LIN {X 0,Y 312.483,Z 284.187,A -85,B 0,C 180,E1 -15707.917,E2 -15707.917} C_VEL
LIN {X 0,Y 312.533,Z 284.181,A -85,B 0,C 180,E1 -15711.909,E2 -15711.909} C_VEL
LIN {X 0,Y 312.504,Z 284.186,A -85,B 0,C 180,E1 -15715.788,E2 -15715.788} C_VEL
LIN {X 0,Y 312.503,Z 284.18,A -85,B 0,C 180,E1 -15718.85,E2 -15718.85} C_VEL
LIN {X 0,Y 312.537,Z 284.181,A -85,B 0,C 180,E1 -15721.82,E2 -15721.82} C_VEL
LIN {X 0,Y 312.544,Z 284.175,A -85,B 0,C 180,E1 -15724.706,E2 -15724.706} C_VEL
LIN {X 0,Y 312.559,Z 284.177,A -85,B 0,C 180,E1 -15727.525,E2 -15727.525} C_VEL
LIN {X 0,Y 312.562,Z 284.179,A -85,B 0,C 180,E1 -15731.65,E2 -15731.65} C_VEL
LIN {X 0,Y 312.68,Z 284.164,A -85,B 0,C 180,E1 -15735.684,E2 -15735.684} C_VEL
LIN {X 0,Y 312.696,Z 284.162,A -85,B 0,C 180,E1 -15739.64,E2 -15739.64} C_VEL
LIN {X 0,Y 312.865,Z 284.136,A -85,B 0,C 180,E1 -15742.252,E2 -15742.252} C_VEL
LIN {X 0,Y 312.708,Z 284.155,A -85,B 0,C 180,E1 -15744.841,E2 -15744.841} C_VEL
LIN {X 0,Y 312.982,Z 284.121,A -85,B 0,C 180,E1 -15748.712,E2 -15748.712} C_VEL
LIN {X 0,Y 312.982,Z 284.123,A -85,B 0,C 180,E1 -15751.285,E2 -15751.285} C_VEL
LIN {X 0,Y 312.707,Z 284.157,A -85,B 0,C 180,E1 -15755.156,E2 -15755.156} C_VEL
LIN {X 0,Y 312.862,Z 284.139,A -85,B 0,C 180,E1 -15757.744,E2 -15757.744} C_VEL
LIN {X 0,Y 312.659,Z 284.164,A -85,B 0,C 180,E1 -15761.67,E2 -15761.67} C_VEL
LIN {X 0,Y 312.69,Z 284.158,A -85,B 0,C 180,E1 -15764.886,E2 -15764.886} C_VEL
LIN {X 0,Y 312.619,Z 284.169,A -85,B 0,C 180,E1 -15769.235,E2 -15769.235} C_VEL
LIN {X 0,Y 312.535,Z 284.177,A -85,B 0,C 180,E1 -15772.788,E2 -15772.788} C_VEL
LIN {X 0,Y 312.585,Z 284.171,A -85,B 0,C 180,E1 -15775.932,E2 -15775.932} C_VEL
LIN {X 0,Y 312.526,Z 284.18,A -85,B 0,C 180,E1 -15779.65,E2 -15779.65} C_VEL
LIN {X 0,Y 312.507,Z 284.182,A -85,B 0,C 180,E1 -15783.688,E2 -15783.688} C_VEL
LIN {X 0,Y 312.525,Z 284.183,A -85,B 0,C 180,E1 -15787.383,E2 -15787.383} C_VEL
LIN {X 0,Y 312.477,Z 284.184,A -85,B 0,C 180,E1 -15790.708,E2 -15790.708} C_VEL
LIN {X 0,Y 312.459,Z 284.185,A -85,B 0,C 180,E1 -15794.205,E2 -15794.205} C_VEL
LIN {X 0,Y 312.472,Z 284.185,A -85,B 0,C 180,E1 -15797.918,E2 -15797.918} C_VEL
LIN {X 0,Y 312.491,Z 284.182,A -85,B 0,C 180,E1 -15801.917,E2 -15801.917} C_VEL
LIN {X 0,Y 312.517,Z 284.178,A -85,B 0,C 180,E1 -15804.22,E2 -15804.22} C_VEL
LIN {X 0,Y 312.49,Z 284.186,A -85,B 0,C 180,E1 -15807.334,E2 -15807.334} C_VEL
LIN {X 0,Y 312.538,Z 284.18,A -85,B 0,C 180,E1 -15811.276,E2 -15811.276} C_VEL
LIN {X 0,Y 312.541,Z 284.176,A -85,B 0,C 180,E1 -15812.722,E2 -15812.722} C_VEL
LIN {X 0,Y 311.9,Z 284.261,A -85,B 0,C 180,E1 -15813.797,E2 -15813.797} C_VEL
LIN {X 0,Y 309.062,Z 284.619,A -85,B 0,C 180,E1 -15815.546,E2 -15815.546} C_VEL
LIN {X 0,Y 306.628,Z 284.92,A -85,B 0,C 180,E1 -15816.965,E2 -15816.965} C_VEL
LIN {X 0,Y 305.562,Z 285.047,A -85,B 0,C 180,E1 -15818.063,E2 -15818.063} C_VEL
LIN {X 0,Y 305.466,Z 285.057,A -85,B 0,C 180,E1 -15818.435,E2 -15818.435} C_VEL
LIN {X 0,Y 305.566,Z 285.049,A -85,B 0,C 180,E1 -15821.217,E2 -15821.217} C_VEL
LIN {X 0,Y 305.635,Z 285.039,A -85,B 0,C 180,E1 -15825.35,E2 -15825.35} C_VEL
LIN {X 0,Y 305.625,Z 285.04,A -85,B 0,C 180,E1 -15829.4,E2 -15829.4} C_VEL
LIN {X 0,Y 305.795,Z 285.016,A -85,B 0,C 180,E1 -15832.075,E2 -15832.075} C_VEL
LIN {X 0,Y 305.673,Z 285.033,A -85,B 0,C 180,E1 -15834.724,E2 -15834.724} C_VEL
LIN {X 0,Y 305.945,Z 284.999,A -85,B 0,C 180,E1 -15838.685,E2 -15838.685} C_VEL
LIN {X 0,Y 305.946,Z 285,A -85,B 0,C 180,E1 -15841.317,E2 -15841.317} C_VEL
LIN {X 0,Y 305.84,Z 285.012,A -85,B 0,C 180,E1 -15846.599,E2 -15846.599} C_VEL
LIN {X 0,Y 305.725,Z 285.027,A -85,B 0,C 180,E1 -15849.261,E2 -15849.261} C_VEL
LIN {X 0,Y 305.578,Z 285.045,A -85,B 0,C 180,E1 -15853.297,E2 -15853.297} C_VEL
LIN {X 0,Y 305.583,Z 285.042,A -85,B 0,C 180,E1 -15856.022,E2 -15856.022} C_VEL
LIN {X 0,Y 305.55,Z 285.048,A -85,B 0,C 180,E1 -15859.438,E2 -15859.438} C_VEL
LIN {X 0,Y 305.476,Z 285.06,A -85,B 0,C 180,E1 -15863.041,E2 -15863.041} C_VEL
LIN {X 0,Y 305.517,Z 285.052,A -85,B 0,C 180,E1 -15866.221,E2 -15866.221} C_VEL
LIN {X 0,Y 305.487,Z 285.058,A -85,B 0,C 180,E1 -15869.052,E2 -15869.052} C_VEL
LIN {X 0,Y 305.457,Z 285.059,A -85,B 0,C 180,E1 -15873.519,E2 -15873.519} C_VEL
LIN {X 0,Y 305.464,Z 285.062,A -85,B 0,C 180,E1 -15876.742,E2 -15876.742} C_VEL
LIN {X 0,Y 305.448,Z 285.063,A -85,B 0,C 180,E1 -15880.602,E2 -15880.602} C_VEL
LIN {X 0,Y 305.413,Z 285.066,A -85,B 0,C 180,E1 -15884.495,E2 -15884.495} C_VEL
LIN {X 0,Y 305.439,Z 285.062,A -85,B 0,C 180,E1 -15888.146,E2 -15888.146} C_VEL
LIN {X 0,Y 305.483,Z 285.18,A -85,B 0,C 180,E1 -15889.323,E2 -15889.323} C_VEL
LIN {X 0,Y 309.162,Z 300.003,A -85,B 0,C 180,E1 -15893.056,E2 -15893.056} C_VEL
LIN {X 0,Y 311.75,Z 310.492,A -85,B 0,C 180,E1 -15895.574,E2 -15895.574} C_VEL
LIN {X 0,Y 318.467,Z 328.782,A -85,B 0,C 180,E1 -15896.765,E2 -15896.765} C_VEL
LIN {X 0,Y 323.204,Z 363.617,A -85,B 0,C 180,E1 -15898.341,E2 -15898.341} C_VEL
LIN {X 0,Y 317.418,Z 478.074,A -85,B 0,C 180,E1 -15901.98,E2 -15901.98} C_VEL
LIN {X 0,Y 316.163,Z 494.683,A -85,B 0,C 180,E1 -15902.769,E2 -15902.769} C_VEL
LIN {X 0,Y 314.676,Z 509.82,A -85,B 0,C 180,E1 -15903.739,E2 -15903.739} C_VEL
LIN {X 0,Y 313.128,Z 524.404,A -85,B 0,C 180,E1 -15904.938,E2 -15904.938} C_VEL
LIN {X 0,Y 311.443,Z 538.622,A -85,B 0,C 180,E1 -15906.39,E2 -15906.39} C_VEL
LIN {X 0,Y 309.762,Z 551.702,A -85,B 0,C 180,E1 -15908.018,E2 -15908.018} C_VEL
LIN {X 0,Y 308.306,Z 563.036,A -85,B 0,C 180,E1 -15909.703,E2 -15909.703} C_VEL
LIN {X 0,Y 306.969,Z 574.069,A -85,B 0,C 180,E1 -15911.653,E2 -15911.653} C_VEL
LIN {X 0,Y 305.696,Z 585.036,A -85,B 0,C 180,E1 -15913.987,E2 -15913.987} C_VEL
LIN {X 0,Y 304.836,Z 594.132,A -85,B 0,C 180,E1 -15916.341,E2 -15916.341} C_VEL
LIN {X 0,Y 304.283,Z 601.551,A -85,B 0,C 180,E1 -15918.68,E2 -15918.68} C_VEL
LIN {X 0,Y 303.985,Z 608.343,A -85,B 0,C 180,E1 -15921.359,E2 -15921.359} C_VEL
LIN {X 0,Y 303.954,Z 613.202,A -85,B 0,C 180,E1 -15923.854,E2 -15923.854} C_VEL
LIN {X 0,Y 303.841,Z 616.375,A -85,B 0,C 180,E1 -15926.023,E2 -15926.023} C_VEL
LIN {X 0,Y 304.058,Z 618.937,A -85,B 0,C 180,E1 -15928.677,E2 -15928.677} C_VEL
LIN {X 0,Y 304.045,Z 619.678,A -85,B 0,C 180,E1 -15930.002,E2 -15930.002} C_VEL
LIN {X 0,Y 303.957,Z 620.077,A -85,B 0,C 180,E1 -15931.327,E2 -15931.327} C_VEL
LIN {X 0,Y 303.763,Z 619.886,A -85,B 0,C 180,E1 -15933.982,E2 -15933.982} C_VEL
LIN {X 0,Y 303.706,Z 618.409,A -85,B 0,C 180,E1 -15936.646,E2 -15936.646} C_VEL
LIN {X 0,Y 303.899,Z 615.68,A -85,B 0,C 180,E1 -15939.318,E2 -15939.318} C_VEL
LIN {X 0,Y 304.501,Z 611.675,A -85,B 0,C 180,E1 -15941.991,E2 -15941.991} C_VEL
LIN {X 0,Y 305.543,Z 606.341,A -85,B 0,C 180,E1 -15944.658,E2 -15944.658} C_VEL
LIN {X 0,Y 307.205,Z 599.572,A -85,B 0,C 180,E1 -15947.303,E2 -15947.303} C_VEL
LIN {X 0,Y 309.461,Z 591.258,A -85,B 0,C 180,E1 -15949.919,E2 -15949.919} C_VEL
LIN {X 0,Y 311.889,Z 582.568,A -85,B 0,C 180,E1 -15952.177,E2 -15952.177} C_VEL
LIN {X 0,Y 315.026,Z 572.349,A -85,B 0,C 180,E1 -15954.378,E2 -15954.378} C_VEL
LIN {X 0,Y 318.596,Z 560.378,A -85,B 0,C 180,E1 -15956.534,E2 -15956.534} C_VEL
LIN {X 0,Y 322.495,Z 547.288,A -85,B 0,C 180,E1 -15958.473,E2 -15958.473} C_VEL
LIN {X 0,Y 326.441,Z 533.561,A -85,B 0,C 180,E1 -15960.143,E2 -15960.143} C_VEL
LIN {X 0,Y 330.508,Z 518.79,A -85,B 0,C 180,E1 -15961.599,E2 -15961.599} C_VEL
LIN {X 0,Y 334.241,Z 504,A -85,B 0,C 180,E1 -15962.783,E2 -15962.783} C_VEL
LIN {X 0,Y 337.95,Z 487.774,A -85,B 0,C 180,E1 -15963.801,E2 -15963.801} C_VEL
LIN {X 0,Y 341.362,Z 470.013,A -85,B 0,C 180,E1 -15964.664,E2 -15964.664} C_VEL
LIN {X 0,Y 353.831,Z 389.949,A -85,B 0,C 180,E1 -15967.737,E2 -15967.737} C_VEL
LIN {X 0,Y 357.008,Z 371.451,A -85,B 0,C 180,E1 -15968.451,E2 -15968.451} C_VEL
LIN {X 0,Y 357.448,Z 364.254,A -85,B 0,C 180,E1 -15969.081,E2 -15969.081} C_VEL
LIN {X 0,Y 356.3,Z 359.523,A -85,B 0,C 180,E1 -15970.263,E2 -15970.263} C_VEL
LIN {X 0,Y 355.233,Z 355.391,A -85,B 0,C 180,E1 -15971.627,E2 -15971.627} C_VEL
LIN {X 0,Y 354.276,Z 351.159,A -85,B 0,C 180,E1 -15973.708,E2 -15973.708} C_VEL
LIN {X 0,Y 354.116,Z 349.484,A -85,B 0,C 180,E1 -15975.187,E2 -15975.187} C_VEL
LIN {X 0,Y 354.487,Z 349.334,A -85,B 0,C 180,E1 -15977.187,E2 -15977.187} C_VEL
LIN {X 0,Y 355.969,Z 350.738,A -85,B 0,C 180,E1 -15979.342,E2 -15979.342} C_VEL
LIN {X 0,Y 357.608,Z 353.477,A -85,B 0,C 180,E1 -15980.911,E2 -15980.911} C_VEL
LIN {X 0,Y 358.995,Z 356.175,A -85,B 0,C 180,E1 -15981.975,E2 -15981.975} C_VEL
LIN {X 0,Y 347.517,Z 422.744,A -85,B 0,C 180,E1 -15984.537,E2 -15984.537} C_VEL
LIN {X 0,Y 342.784,Z 453.541,A -85,B 0,C 180,E1 -15985.767,E2 -15985.767} C_VEL
LIN {X 0,Y 339.824,Z 469.984,A -85,B 0,C 180,E1 -15986.677,E2 -15986.677} C_VEL
LIN {X 0,Y 336.515,Z 485.723,A -85,B 0,C 180,E1 -15987.821,E2 -15987.821} C_VEL
LIN {X 0,Y 333.231,Z 499.427,A -85,B 0,C 180,E1 -15989.063,E2 -15989.063} C_VEL
LIN {X 0,Y 329.525,Z 513.47,A -85,B 0,C 180,E1 -15990.623,E2 -15990.623} C_VEL
LIN {X 0,Y 325.894,Z 525.991,A -85,B 0,C 180,E1 -15992.318,E2 -15992.318} C_VEL
LIN {X 0,Y 322.284,Z 537.29,A -85,B 0,C 180,E1 -15994.142,E2 -15994.142} C_VEL
LIN {X 0,Y 318.668,Z 548.098,A -85,B 0,C 180,E1 -15996.265,E2 -15996.265} C_VEL
LIN {X 0,Y 315.639,Z 557.162,A -85,B 0,C 180,E1 -15998.445,E2 -15998.445} C_VEL
LIN {X 0,Y 312.714,Z 565.295,A -85,B 0,C 180,E1 -16000.805,E2 -16000.805} C_VEL
LIN {X 0,Y 310.44,Z 571.206,A -85,B 0,C 180,E1 -16002.883,E2 -16002.883} C_VEL
LIN {X 0,Y 308.415,Z 577.037,A -85,B 0,C 180,E1 -16005.482,E2 -16005.482} C_VEL
LIN {X 0,Y 306.824,Z 581.492,A -85,B 0,C 180,E1 -16008.102,E2 -16008.102} C_VEL
LIN {X 0,Y 305.638,Z 584.662,A -85,B 0,C 180,E1 -16010.736,E2 -16010.736} C_VEL
LIN {X 0,Y 304.678,Z 586.616,A -85,B 0,C 180,E1 -16013.376,E2 -16013.376} C_VEL
LIN {X 0,Y 304.271,Z 587.337,A -85,B 0,C 180,E1 -16016.026,E2 -16016.026} C_VEL
LIN {X 0,Y 303.995,Z 586.847,A -85,B 0,C 180,E1 -16018.674,E2 -16018.674} C_VEL
LIN {X 0,Y 303.845,Z 585.118,A -85,B 0,C 180,E1 -16021.324,E2 -16021.324} C_VEL
LIN {X 0,Y 303.946,Z 582.089,A -85,B 0,C 180,E1 -16023.977,E2 -16023.977} C_VEL
LIN {X 0,Y 304.108,Z 577.7,A -85,B 0,C 180,E1 -16026.634,E2 -16026.634} C_VEL
LIN {X 0,Y 304.48,Z 571.858,A -85,B 0,C 180,E1 -16029.297,E2 -16029.297} C_VEL
LIN {X 0,Y 305.091,Z 564.369,A -85,B 0,C 180,E1 -16031.964,E2 -16031.964} C_VEL
LIN {X 0,Y 306.037,Z 556.302,A -85,B 0,C 180,E1 -16034.291,E2 -16034.291} C_VEL
LIN {X 0,Y 307.118,Z 546.548,A -85,B 0,C 180,E1 -16036.62,E2 -16036.62} C_VEL
LIN {X 0,Y 308.375,Z 536.618,A -85,B 0,C 180,E1 -16038.605,E2 -16038.605} C_VEL
LIN {X 0,Y 309.868,Z 524.859,A -85,B 0,C 180,E1 -16040.581,E2 -16040.581} C_VEL
LIN {X 0,Y 311.38,Z 512.154,A -85,B 0,C 180,E1 -16042.363,E2 -16042.363} C_VEL
LIN {X 0,Y 312.995,Z 497.882,A -85,B 0,C 180,E1 -16044.014,E2 -16044.014} C_VEL
LIN {X 0,Y 314.43,Z 484.235,A -85,B 0,C 180,E1 -16045.306,E2 -16045.306} C_VEL
LIN {X 0,Y 315.759,Z 469.495,A -85,B 0,C 180,E1 -16046.431,E2 -16046.431} C_VEL
LIN {X 0,Y 316.948,Z 453.178,A -85,B 0,C 180,E1 -16047.392,E2 -16047.392} C_VEL
LIN {X 0,Y 317.883,Z 437.277,A -85,B 0,C 180,E1 -16048.065,E2 -16048.065} C_VEL
LIN {X 0,Y 323.396,Z 326.411,A -85,B 0,C 180,E1 -16051.547,E2 -16051.547} C_VEL
LIN {X 0,Y 307.407,Z 290.038,A -85,B 0,C 180,E1 -16054.103,E2 -16054.103} C_VEL
LIN {X 0,Y 305.517,Z 285.343,A -85,B 0,C 180,E1 -16054.439,E2 -16054.439} C_VEL
LIN {X 0,Y 305.491,Z 285.056,A -85,B 0,C 180,E1 -16054.482,E2 -16054.482} C_VEL
LIN {X 0,Y 305.427,Z 285.063,A -85,B 0,C 180,E1 -16058.521,E2 -16058.521} C_VEL
LIN {X 0,Y 305.439,Z 285.066,A -85,B 0,C 180,E1 -16061.855,E2 -16061.855} C_VEL
LIN {X 0,Y 305.399,Z 285.068,A -85,B 0,C 180,E1 -16065.509,E2 -16065.509} C_VEL
LIN {X 0,Y 305.44,Z 285.063,A -85,B 0,C 180,E1 -16068.141,E2 -16068.141} C_VEL
LIN {X 0,Y 305.493,Z 285.057,A -85,B 0,C 180,E1 -16071.598,E2 -16071.598} C_VEL
LIN {X 0,Y 305.46,Z 285.058,A -85,B 0,C 180,E1 -16074.885,E2 -16074.885} C_VEL
LIN {X 0,Y 305.438,Z 285.061,A -85,B 0,C 180,E1 -16078.356,E2 -16078.356} C_VEL
LIN {X 0,Y 305.482,Z 285.056,A -85,B 0,C 180,E1 -16081.108,E2 -16081.108} C_VEL
LIN {X 0,Y 305.497,Z 285.055,A -85,B 0,C 180,E1 -16084.08,E2 -16084.08} C_VEL
LIN {X 0,Y 305.488,Z 285.055,A -85,B 0,C 180,E1 -16086.975,E2 -16086.975} C_VEL
LIN {X 0,Y 305.513,Z 285.053,A -85,B 0,C 180,E1 -16091.211,E2 -16091.211} C_VEL
LIN {X 0,Y 305.621,Z 285.041,A -85,B 0,C 180,E1 -16095.346,E2 -16095.346} C_VEL
LIN {X 0,Y 305.632,Z 285.04,A -85,B 0,C 180,E1 -16099.398,E2 -16099.398} C_VEL
LIN {X 0,Y 305.806,Z 285.016,A -85,B 0,C 180,E1 -16102.072,E2 -16102.072} C_VEL
LIN {X 0,Y 305.68,Z 285.03,A -85,B 0,C 180,E1 -16104.722,E2 -16104.722} C_VEL
LIN {X 0,Y 305.949,Z 284.997,A -85,B 0,C 180,E1 -16108.682,E2 -16108.682} C_VEL
LIN {X 0,Y 305.949,Z 285,A -85,B 0,C 180,E1 -16111.314,E2 -16111.314} C_VEL
LIN {X 0,Y 305.843,Z 285.01,A -85,B 0,C 180,E1 -16116.596,E2 -16116.596} C_VEL
LIN {X 0,Y 305.727,Z 285.027,A -85,B 0,C 180,E1 -16119.258,E2 -16119.258} C_VEL
LIN {X 0,Y 305.579,Z 285.046,A -85,B 0,C 180,E1 -16123.294,E2 -16123.294} C_VEL
LIN {X 0,Y 305.583,Z 285.043,A -85,B 0,C 180,E1 -16126.019,E2 -16126.019} C_VEL
LIN {X 0,Y 305.566,Z 285.049,A -85,B 0,C 180,E1 -16129.443,E2 -16129.443} C_VEL
LIN {X 0,Y 305.479,Z 285.057,A -85,B 0,C 180,E1 -16133.04,E2 -16133.04} C_VEL
LIN {X 0,Y 305.514,Z 285.051,A -85,B 0,C 180,E1 -16136.217,E2 -16136.217} C_VEL
LIN {X 0,Y 305.476,Z 285.058,A -85,B 0,C 180,E1 -16139.046,E2 -16139.046} C_VEL
LIN {X 0,Y 305.429,Z 285.062,A -85,B 0,C 180,E1 -16141.951,E2 -16141.951} C_VEL
LIN {X 0,Y 305.45,Z 285.062,A -85,B 0,C 180,E1 -16145.112,E2 -16145.112} C_VEL
LIN {X 0,Y 305.436,Z 285.061,A -85,B 0,C 180,E1 -16148.528,E2 -16148.528} C_VEL
LIN {X 0,Y 305.446,Z 285.06,A -85,B 0,C 180,E1 -16152.586,E2 -16152.586} C_VEL
LIN {X 0,Y 305.429,Z 285.061,A -85,B 0,C 180,E1 -16156.347,E2 -16156.347} C_VEL
LIN {X 0,Y 305.444,Z 285.06,A -85,B 0,C 180,E1 -16159.892,E2 -16159.892} C_VEL
LIN {X 0,Y 305.467,Z 285.059,A -85,B 0,C 180,E1 -16163.631,E2 -16163.631} C_VEL
LIN {X 0,Y 305.451,Z 285.059,A -85,B 0,C 180,E1 -16166.483,E2 -16166.483} C_VEL
LIN {X 0,Y 305.482,Z 285.058,A -85,B 0,C 180,E1 -16170.95,E2 -16170.95} C_VEL
LIN {X 0,Y 305.558,Z 285.045,A -85,B 0,C 180,E1 -16174.088,E2 -16174.088} C_VEL
LIN {X 0,Y 305.466,Z 285.057,A -85,B 0,C 180,E1 -16178.435,E2 -16178.435} C_VEL
LIN {X 0,Y 304.775,Z 285.145,A -85,B 0,C 180,E1 -16179.537,E2 -16179.537} C_VEL
LIN {X 0,Y 301.943,Z 285.499,A -85,B 0,C 180,E1 -16181.332,E2 -16181.332} C_VEL
LIN {X 0,Y 299.585,Z 285.792,A -85,B 0,C 180,E1 -16182.788,E2 -16182.788} C_VEL
LIN {X 0,Y 298.613,Z 285.911,A -85,B 0,C 180,E1 -16183.915,E2 -16183.915} C_VEL
LIN {X 0,Y 298.553,Z 285.918,A -85,B 0,C 180,E1 -16184.296,E2 -16184.296} C_VEL
LIN {X 0,Y 298.54,Z 285.919,A -85,B 0,C 180,E1 -16187.769,E2 -16187.769} C_VEL
LIN {X 0,Y 298.741,Z 285.895,A -85,B 0,C 180,E1 -16191.887,E2 -16191.887} C_VEL
LIN {X 0,Y 298.644,Z 285.908,A -85,B 0,C 180,E1 -16194.6,E2 -16194.6} C_VEL
LIN {X 0,Y 298.911,Z 285.875,A -85,B 0,C 180,E1 -16198.654,E2 -16198.654} C_VEL
LIN {X 0,Y 298.913,Z 285.875,A -85,B 0,C 180,E1 -16201.348,E2 -16201.348} C_VEL
LIN {X 0,Y 298.785,Z 285.892,A -85,B 0,C 180,E1 -16206.755,E2 -16206.755} C_VEL
LIN {X 0,Y 298.67,Z 285.905,A -85,B 0,C 180,E1 -16209.482,E2 -16209.482} C_VEL
LIN {X 0,Y 298.541,Z 285.92,A -85,B 0,C 180,E1 -16213.617,E2 -16213.617} C_VEL
LIN {X 0,Y 298.538,Z 285.921,A -85,B 0,C 180,E1 -16216.41,E2 -16216.41} C_VEL
LIN {X 0,Y 298.488,Z 285.927,A -85,B 0,C 180,E1 -16219.649,E2 -16219.649} C_VEL
LIN {X 0,Y 298.419,Z 285.936,A -85,B 0,C 180,E1 -16223.602,E2 -16223.602} C_VEL
LIN {X 0,Y 298.477,Z 285.931,A -85,B 0,C 180,E1 -16226.577,E2 -16226.577} C_VEL
LIN {X 0,Y 298.412,Z 285.936,A -85,B 0,C 180,E1 -16229.643,E2 -16229.643} C_VEL
LIN {X 0,Y 298.387,Z 285.944,A -85,B 0,C 180,E1 -16232.802,E2 -16232.802} C_VEL
LIN {X 0,Y 298.436,Z 285.938,A -85,B 0,C 180,E1 -16236.809,E2 -16236.809} C_VEL
LIN {X 0,Y 298.381,Z 285.942,A -85,B 0,C 180,E1 -16241.09,E2 -16241.09} C_VEL
LIN {X 0,Y 298.383,Z 285.942,A -85,B 0,C 180,E1 -16245.044,E2 -16245.044} C_VEL
LIN {X 0,Y 298.417,Z 286.041,A -85,B 0,C 180,E1 -16248.854,E2 -16248.854} C_VEL
LIN {X 0,Y 302.253,Z 301.368,A -85,B 0,C 180,E1 -16252.806,E2 -16252.806} C_VEL
LIN {X 0,Y 304.389,Z 310.097,A -85,B 0,C 180,E1 -16254.948,E2 -16254.948} C_VEL
LIN {X 0,Y 312.03,Z 331.055,A -85,B 0,C 180,E1 -16256.362,E2 -16256.362} C_VEL
LIN {X 0,Y 316.55,Z 364.738,A -85,B 0,C 180,E1 -16257.919,E2 -16257.919} C_VEL
LIN {X 0,Y 310.599,Z 477.927,A -85,B 0,C 180,E1 -16261.632,E2 -16261.632} C_VEL
LIN {X 0,Y 309.42,Z 493.04,A -85,B 0,C 180,E1 -16262.354,E2 -16262.354} C_VEL
LIN {X 0,Y 307.855,Z 508.932,A -85,B 0,C 180,E1 -16263.386,E2 -16263.386} C_VEL
LIN {X 0,Y 306.165,Z 524.431,A -85,B 0,C 180,E1 -16264.691,E2 -16264.691} C_VEL
LIN {X 0,Y 304.46,Z 538.557,A -85,B 0,C 180,E1 -16266.176,E2 -16266.176} C_VEL
LIN {X 0,Y 302.736,Z 551.563,A -85,B 0,C 180,E1 -16267.839,E2 -16267.839} C_VEL
LIN {X 0,Y 301.165,Z 563.609,A -85,B 0,C 180,E1 -16269.691,E2 -16269.691} C_VEL
LIN {X 0,Y 299.892,Z 573.843,A -85,B 0,C 180,E1 -16271.558,E2 -16271.558} C_VEL
LIN {X 0,Y 298.631,Z 584.784,A -85,B 0,C 180,E1 -16273.949,E2 -16273.949} C_VEL
LIN {X 0,Y 297.738,Z 593.823,A -85,B 0,C 180,E1 -16276.349,E2 -16276.349} C_VEL
LIN {X 0,Y 297.273,Z 600.297,A -85,B 0,C 180,E1 -16278.409,E2 -16278.409} C_VEL
LIN {X 0,Y 296.919,Z 607.265,A -85,B 0,C 180,E1 -16281.152,E2 -16281.152} C_VEL
LIN {X 0,Y 296.9,Z 612.479,A -85,B 0,C 180,E1 -16283.827,E2 -16283.827} C_VEL
LIN {X 0,Y 296.781,Z 615.545,A -85,B 0,C 180,E1 -16285.928,E2 -16285.928} C_VEL
LIN {X 0,Y 296.999,Z 618.242,A -85,B 0,C 180,E1 -16288.646,E2 -16288.646} C_VEL
LIN {X 0,Y 296.991,Z 619.051,A -85,B 0,C 180,E1 -16290.002,E2 -16290.002} C_VEL
LIN {X 0,Y 296.881,Z 619.516,A -85,B 0,C 180,E1 -16291.358,E2 -16291.358} C_VEL
LIN {X 0,Y 296.668,Z 619.463,A -85,B 0,C 180,E1 -16294.077,E2 -16294.077} C_VEL
LIN {X 0,Y 296.623,Z 618.133,A -85,B 0,C 180,E1 -16296.805,E2 -16296.805} C_VEL
LIN {X 0,Y 296.835,Z 615.553,A -85,B 0,C 180,E1 -16299.542,E2 -16299.542} C_VEL
LIN {X 0,Y 297.515,Z 611.694,A -85,B 0,C 180,E1 -16302.277,E2 -16302.277} C_VEL
LIN {X 0,Y 298.827,Z 605.745,A -85,B 0,C 180,E1 -16305.362,E2 -16305.362} C_VEL
LIN {X 0,Y 300.968,Z 598.071,A -85,B 0,C 180,E1 -16308.377,E2 -16308.377} C_VEL
LIN {X 0,Y 303.498,Z 589.608,A -85,B 0,C 180,E1 -16311.036,E2 -16311.036} C_VEL
LIN {X 0,Y 306.3,Z 580.882,A -85,B 0,C 180,E1 -16313.3,E2 -16313.3} C_VEL
LIN {X 0,Y 309.65,Z 570.511,A -85,B 0,C 180,E1 -16315.548,E2 -16315.548} C_VEL
LIN {X 0,Y 313.615,Z 558.405,A -85,B 0,C 180,E1 -16317.712,E2 -16317.712} C_VEL
LIN {X 0,Y 317.865,Z 545.2,A -85,B 0,C 180,E1 -16319.652,E2 -16319.652} C_VEL
LIN {X 0,Y 322.293,Z 530.854,A -85,B 0,C 180,E1 -16321.376,E2 -16321.376} C_VEL
LIN {X 0,Y 326.852,Z 515.219,A -85,B 0,C 180,E1 -16322.885,E2 -16322.885} C_VEL
LIN {X 0,Y 330.484,Z 501.733,A -85,B 0,C 180,E1 -16323.935,E2 -16323.935} C_VEL
LIN {X 0,Y 334.701,Z 484.374,A -85,B 0,C 180,E1 -16324.996,E2 -16324.996} C_VEL
LIN {X 0,Y 338.319,Z 465.747,A -85,B 0,C 180,E1 -16325.881,E2 -16325.881} C_VEL
LIN {X 0,Y 350.487,Z 393.563,A -85,B 0,C 180,E1 -16328.663,E2 -16328.663} C_VEL
LIN {X 0,Y 354.184,Z 373.355,A -85,B 0,C 180,E1 -16329.461,E2 -16329.461} C_VEL
LIN {X 0,Y 354.573,Z 368.802,A -85,B 0,C 180,E1 -16329.869,E2 -16329.869} C_VEL
LIN {X 0,Y 353.784,Z 365.071,A -85,B 0,C 180,E1 -16330.872,E2 -16330.872} C_VEL
LIN {X 0,Y 353.025,Z 361.495,A -85,B 0,C 180,E1 -16332.093,E2 -16332.093} C_VEL
LIN {X 0,Y 352.349,Z 357.579,A -85,B 0,C 180,E1 -16334.105,E2 -16334.105} C_VEL
LIN {X 0,Y 352.304,Z 356.267,A -85,B 0,C 180,E1 -16335.371,E2 -16335.371} C_VEL
LIN {X 0,Y 352.911,Z 356.433,A -85,B 0,C 180,E1 -16337.679,E2 -16337.679} C_VEL
LIN {X 0,Y 354.031,Z 357.544,A -85,B 0,C 180,E1 -16339.218,E2 -16339.218} C_VEL
LIN {X 0,Y 355.445,Z 360.103,A -85,B 0,C 180,E1 -16340.68,E2 -16340.68} C_VEL
LIN {X 0,Y 355.888,Z 361.083,A -85,B 0,C 180,E1 -16341.077,E2 -16341.077} C_VEL
LIN {X 0,Y 342.922,Z 431.583,A -85,B 0,C 180,E1 -16343.807,E2 -16343.807} C_VEL
LIN {X 0,Y 339.137,Z 454.518,A -85,B 0,C 180,E1 -16344.759,E2 -16344.759} C_VEL
LIN {X 0,Y 336.129,Z 470.041,A -85,B 0,C 180,E1 -16345.629,E2 -16345.629} C_VEL
LIN {X 0,Y 332.763,Z 484.823,A -85,B 0,C 180,E1 -16346.692,E2 -16346.692} C_VEL
LIN {X 0,Y 329.231,Z 498.567,A -85,B 0,C 180,E1 -16347.926,E2 -16347.926} C_VEL
LIN {X 0,Y 324.919,Z 513.833,A -85,B 0,C 180,E1 -16349.628,E2 -16349.628} C_VEL
LIN {X 0,Y 320.652,Z 527.393,A -85,B 0,C 180,E1 -16351.498,E2 -16351.498} C_VEL
LIN {X 0,Y 316.277,Z 539.949,A -85,B 0,C 180,E1 -16353.613,E2 -16353.613} C_VEL
LIN {X 0,Y 312.51,Z 550.345,A -85,B 0,C 180,E1 -16355.768,E2 -16355.768} C_VEL
LIN {X 0,Y 309.285,Z 559.083,A -85,B 0,C 180,E1 -16357.979,E2 -16357.979} C_VEL
LIN {X 0,Y 306.542,Z 566.186,A -85,B 0,C 180,E1 -16360.133,E2 -16360.133} C_VEL
LIN {X 0,Y 303.821,Z 572.657,A -85,B 0,C 180,E1 -16362.498,E2 -16362.498} C_VEL
LIN {X 0,Y 301.654,Z 578.271,A -85,B 0,C 180,E1 -16365.15,E2 -16365.15} C_VEL
LIN {X 0,Y 300.623,Z 580.589,A -85,B 0,C 180,E1 -16366.479,E2 -16366.479} C_VEL
LIN {X 0,Y 299.323,Z 584.168,A -85,B 0,C 180,E1 -16369.172,E2 -16369.172} C_VEL
LIN {X 0,Y 298.052,Z 586.676,A -85,B 0,C 180,E1 -16372.042,E2 -16372.042} C_VEL
LIN {X 0,Y 297.336,Z 587.72,A -85,B 0,C 180,E1 -16374.574,E2 -16374.574} C_VEL
LIN {X 0,Y 297.084,Z 587.662,A -85,B 0,C 180,E1 -16377.287,E2 -16377.287} C_VEL
LIN {X 0,Y 296.779,Z 586.396,A -85,B 0,C 180,E1 -16379.999,E2 -16379.999} C_VEL
LIN {X 0,Y 296.789,Z 583.869,A -85,B 0,C 180,E1 -16382.713,E2 -16382.713} C_VEL
LIN {X 0,Y 296.892,Z 580.019,A -85,B 0,C 180,E1 -16385.432,E2 -16385.432} C_VEL
LIN {X 0,Y 297.208,Z 574.747,A -85,B 0,C 180,E1 -16388.156,E2 -16388.156} C_VEL
LIN {X 0,Y 297.707,Z 567.894,A -85,B 0,C 180,E1 -16390.885,E2 -16390.885} C_VEL
LIN {X 0,Y 298.548,Z 560.487,A -85,B 0,C 180,E1 -16393.268,E2 -16393.268} C_VEL
LIN {X 0,Y 299.466,Z 551.583,A -85,B 0,C 180,E1 -16395.635,E2 -16395.635} C_VEL
LIN {X 0,Y 300.618,Z 542.368,A -85,B 0,C 180,E1 -16397.692,E2 -16397.692} C_VEL
LIN {X 0,Y 302.101,Z 530.593,A -85,B 0,C 180,E1 -16399.89,E2 -16399.89} C_VEL
LIN {X 0,Y 303.625,Z 518.734,A -85,B 0,C 180,E1 -16401.736,E2 -16401.736} C_VEL
LIN {X 0,Y 305.143,Z 505.928,A -85,B 0,C 180,E1 -16403.408,E2 -16403.408} C_VEL
LIN {X 0,Y 306.732,Z 492.126,A -85,B 0,C 180,E1 -16404.897,E2 -16404.897} C_VEL
LIN {X 0,Y 308.216,Z 477.044,A -85,B 0,C 180,E1 -16406.217,E2 -16406.217} C_VEL
LIN {X 0,Y 309.549,Z 461.608,A -85,B 0,C 180,E1 -16407.278,E2 -16407.278} C_VEL
LIN {X 0,Y 310.631,Z 444.902,A -85,B 0,C 180,E1 -16408.141,E2 -16408.141} C_VEL
LIN {X 0,Y 312.036,Z 417.268,A -85,B 0,C 180,E1 -16409.1,E2 -16409.1} C_VEL
LIN {X 0,Y 316.726,Z 328.239,A -85,B 0,C 180,E1 -16411.959,E2 -16411.959} C_VEL
LIN {X 0,Y 300.708,Z 291.611,A -85,B 0,C 180,E1 -16414.6,E2 -16414.6} C_VEL
LIN {X 0,Y 298.508,Z 286.374,A -85,B 0,C 180,E1 -16414.989,E2 -16414.989} C_VEL
LIN {X 0,Y 298.427,Z 285.935,A -85,B 0,C 180,E1 -16415.017,E2 -16415.017} C_VEL
LIN {X 0,Y 298.391,Z 285.94,A -85,B 0,C 180,E1 -16418.988,E2 -16418.988} C_VEL
LIN {X 0,Y 298.399,Z 285.938,A -85,B 0,C 180,E1 -16423.101,E2 -16423.101} C_VEL
LIN {X 0,Y 298.402,Z 285.937,A -85,B 0,C 180,E1 -16426.919,E2 -16426.919} C_VEL
LIN {X 0,Y 298.413,Z 285.935,A -85,B 0,C 180,E1 -16431.002,E2 -16431.002} C_VEL
LIN {X 0,Y 298.417,Z 285.939,A -85,B 0,C 180,E1 -16433.928,E2 -16433.928} C_VEL
LIN {X 0,Y 298.385,Z 285.942,A -85,B 0,C 180,E1 -16437.984,E2 -16437.984} C_VEL
LIN {X 0,Y 298.417,Z 285.939,A -85,B 0,C 180,E1 -16441.898,E2 -16441.898} C_VEL
LIN {X 0,Y 298.437,Z 285.933,A -85,B 0,C 180,E1 -16444.918,E2 -16444.918} C_VEL
LIN {X 0,Y 298.41,Z 285.94,A -85,B 0,C 180,E1 -16447.861,E2 -16447.861} C_VEL
LIN {X 0,Y 298.473,Z 285.928,A -85,B 0,C 180,E1 -16450.751,E2 -16450.751} C_VEL
LIN {X 0,Y 298.58,Z 285.916,A -85,B 0,C 180,E1 -16454.992,E2 -16454.992} C_VEL
LIN {X 0,Y 298.588,Z 285.915,A -85,B 0,C 180,E1 -16459.145,E2 -16459.145} C_VEL
LIN {X 0,Y 298.752,Z 285.896,A -85,B 0,C 180,E1 -16461.884,E2 -16461.884} C_VEL
LIN {X 0,Y 298.651,Z 285.905,A -85,B 0,C 180,E1 -16464.597,E2 -16464.597} C_VEL
LIN {X 0,Y 298.916,Z 285.873,A -85,B 0,C 180,E1 -16468.651,E2 -16468.651} C_VEL
LIN {X 0,Y 298.915,Z 285.876,A -85,B 0,C 180,E1 -16471.345,E2 -16471.345} C_VEL
LIN {X 0,Y 298.788,Z 285.889,A -85,B 0,C 180,E1 -16476.752,E2 -16476.752} C_VEL
LIN {X 0,Y 298.671,Z 285.908,A -85,B 0,C 180,E1 -16479.479,E2 -16479.479} C_VEL
LIN {X 0,Y 298.542,Z 285.923,A -85,B 0,C 180,E1 -16483.614,E2 -16483.614} C_VEL
LIN {X 0,Y 298.538,Z 285.92,A -85,B 0,C 180,E1 -16486.407,E2 -16486.407} C_VEL
LIN {X 0,Y 298.501,Z 285.928,A -85,B 0,C 180,E1 -16489.653,E2 -16489.653} C_VEL
LIN {X 0,Y 298.446,Z 285.935,A -85,B 0,C 180,E1 -16493.596,E2 -16493.596} C_VEL
LIN {X 0,Y 298.473,Z 285.927,A -85,B 0,C 180,E1 -16496.574,E2 -16496.574} C_VEL
LIN {X 0,Y 298.404,Z 285.94,A -85,B 0,C 180,E1 -16499.64,E2 -16499.64} C_VEL
LIN {X 0,Y 298.382,Z 285.94,A -85,B 0,C 180,E1 -16502.799,E2 -16502.799} C_VEL
LIN {X 0,Y 298.452,Z 285.931,A -85,B 0,C 180,E1 -16506.811,E2 -16506.811} C_VEL
LIN {X 0,Y 298.375,Z 285.944,A -85,B 0,C 180,E1 -16511.087,E2 -16511.087} C_VEL
LIN {X 0,Y 298.375,Z 285.943,A -85,B 0,C 180,E1 -16515.041,E2 -16515.041} C_VEL
LIN {X 0,Y 298.374,Z 285.943,A -85,B 0,C 180,E1 -16518.912,E2 -16518.912} C_VEL
LIN {X 0,Y 298.432,Z 285.937,A -85,B 0,C 180,E1 -16523.192,E2 -16523.192} C_VEL
LIN {X 0,Y 298.381,Z 285.945,A -85,B 0,C 180,E1 -16527.2,E2 -16527.2} C_VEL
LIN {X 0,Y 298.455,Z 285.93,A -85,B 0,C 180,E1 -16531.905,E2 -16531.905} C_VEL
LIN {X 0,Y 298.47,Z 285.931,A -85,B 0,C 180,E1 -16534.924,E2 -16534.924} C_VEL
LIN {X 0,Y 298.423,Z 285.937,A -85,B 0,C 180,E1 -16539.315,E2 -16539.315} C_VEL
LIN {X 0,Y 298.521,Z 285.922,A -85,B 0,C 180,E1 -16542.18,E2 -16542.18} C_VEL
LIN {X 0,Y 298.553,Z 285.918,A -85,B 0,C 180,E1 -16544.296,E2 -16544.296} C_VEL
LIN {X 0,Y 297.92,Z 286.001,A -85,B 0,C 180,E1 -16545.422,E2 -16545.422} C_VEL
LIN {X 0,Y 295.038,Z 286.359,A -85,B 0,C 180,E1 -16547.253,E2 -16547.253} C_VEL
LIN {X 0,Y 292.619,Z 286.659,A -85,B 0,C 180,E1 -16548.74,E2 -16548.74} C_VEL
LIN {X 0,Y 291.653,Z 286.777,A -85,B 0,C 180,E1 -16549.893,E2 -16549.893} C_VEL
LIN {X 0,Y 291.616,Z 286.782,A -85,B 0,C 180,E1 -16550.283,E2 -16550.283} C_VEL
LIN {X 0,Y 291.728,Z 286.773,A -85,B 0,C 180,E1 -16553.083,E2 -16553.083} C_VEL
LIN {X 0,Y 291.877,Z 286.751,A -85,B 0,C 180,E1 -16558.621,E2 -16558.621} C_VEL
LIN {X 0,Y 291.879,Z 286.751,A -85,B 0,C 180,E1 -16561.381,E2 -16561.381} C_VEL
LIN {X 0,Y 291.734,Z 286.772,A -85,B 0,C 180,E1 -16566.919,E2 -16566.919} C_VEL
LIN {X 0,Y 291.618,Z 286.782,A -85,B 0,C 180,E1 -16569.713,E2 -16569.713} C_VEL
LIN {X 0,Y 291.511,Z 286.795,A -85,B 0,C 180,E1 -16573.952,E2 -16573.952} C_VEL
LIN {X 0,Y 291.476,Z 286.804,A -85,B 0,C 180,E1 -16576.819,E2 -16576.819} C_VEL
LIN {X 0,Y 291.441,Z 286.805,A -85,B 0,C 180,E1 -16579.876,E2 -16579.876} C_VEL
LIN {X 0,Y 291.373,Z 286.814,A -85,B 0,C 180,E1 -16584.209,E2 -16584.209} C_VEL
LIN {X 0,Y 291.412,Z 286.81,A -85,B 0,C 180,E1 -16587.274,E2 -16587.274} C_VEL
LIN {X 0,Y 291.329,Z 286.82,A -85,B 0,C 180,E1 -16590.439,E2 -16590.439} C_VEL
LIN {X 0,Y 291.337,Z 286.817,A -85,B 0,C 180,E1 -16593.7,E2 -16593.7} C_VEL
LIN {X 0,Y 291.364,Z 286.815,A -85,B 0,C 180,E1 -16597.255,E2 -16597.255} C_VEL
LIN {X 0,Y 291.326,Z 286.822,A -85,B 0,C 180,E1 -16600.645,E2 -16600.645} C_VEL
LIN {X 0,Y 291.308,Z 286.822,A -85,B 0,C 180,E1 -16604.399,E2 -16604.399} C_VEL
LIN {X 0,Y 291.373,Z 286.986,A -85,B 0,C 180,E1 -16608.395,E2 -16608.395} C_VEL
LIN {X 0,Y 294.673,Z 300.256,A -85,B 0,C 180,E1 -16611.912,E2 -16611.912} C_VEL
LIN {X 0,Y 297.094,Z 310.039,A -85,B 0,C 180,E1 -16614.335,E2 -16614.335} C_VEL
LIN {X 0,Y 305.693,Z 333.545,A -85,B 0,C 180,E1 -16615.958,E2 -16615.958} C_VEL
LIN {X 0,Y 309.93,Z 365.207,A -85,B 0,C 180,E1 -16617.468,E2 -16617.468} C_VEL
LIN {X 0,Y 303.787,Z 477.457,A -85,B 0,C 180,E1 -16621.267,E2 -16621.267} C_VEL
LIN {X 0,Y 302.549,Z 492.906,A -85,B 0,C 180,E1 -16622.03,E2 -16622.03} C_VEL
LIN {X 0,Y 300.928,Z 508.903,A -85,B 0,C 180,E1 -16623.099,E2 -16623.099} C_VEL
LIN {X 0,Y 299.2,Z 524.312,A -85,B 0,C 180,E1 -16624.432,E2 -16624.432} C_VEL
LIN {X 0,Y 297.464,Z 538.387,A -85,B 0,C 180,E1 -16625.951,E2 -16625.951} C_VEL
LIN {X 0,Y 295.722,Z 551.359,A -85,B 0,C 180,E1 -16627.653,E2 -16627.653} C_VEL
LIN {X 0,Y 294.001,Z 564.377,A -85,B 0,C 180,E1 -16629.722,E2 -16629.722} C_VEL
LIN {X 0,Y 292.651,Z 575.28,A -85,B 0,C 180,E1 -16631.811,E2 -16631.811} C_VEL
LIN {X 0,Y 291.566,Z 584.485,A -85,B 0,C 180,E1 -16633.909,E2 -16633.909} C_VEL
LIN {X 0,Y 290.658,Z 593.499,A -85,B 0,C 180,E1 -16636.366,E2 -16636.366} C_VEL
LIN {X 0,Y 290.106,Z 600.903,A -85,B 0,C 180,E1 -16638.827,E2 -16638.827} C_VEL
LIN {X 0,Y 289.856,Z 607.653,A -85,B 0,C 180,E1 -16641.637,E2 -16641.637} C_VEL
LIN {X 0,Y 289.867,Z 612.741,A -85,B 0,C 180,E1 -16644.437,E2 -16644.437} C_VEL
LIN {X 0,Y 289.739,Z 616.271,A -85,B 0,C 180,E1 -16647.221,E2 -16647.221} C_VEL
LIN {X 0,Y 289.941,Z 617.526,A -85,B 0,C 180,E1 -16648.613,E2 -16648.613} C_VEL
LIN {X 0,Y 289.938,Z 618.412,A -85,B 0,C 180,E1 -16650.002,E2 -16650.002} C_VEL
LIN {X 0,Y 289.808,Z 618.948,A -85,B 0,C 180,E1 -16651.391,E2 -16651.391} C_VEL
LIN {X 0,Y 289.578,Z 619.043,A -85,B 0,C 180,E1 -16654.177,E2 -16654.177} C_VEL
LIN {X 0,Y 289.542,Z 617.863,A -85,B 0,C 180,E1 -16656.973,E2 -16656.973} C_VEL
LIN {X 0,Y 289.761,Z 615.397,A -85,B 0,C 180,E1 -16659.777,E2 -16659.777} C_VEL
LIN {X 0,Y 290.508,Z 611.685,A -85,B 0,C 180,E1 -16662.577,E2 -16662.577} C_VEL
LIN {X 0,Y 291.867,Z 606.239,A -85,B 0,C 180,E1 -16665.595,E2 -16665.595} C_VEL
LIN {X 0,Y 293.625,Z 600.358,A -85,B 0,C 180,E1 -16668.131,E2 -16668.131} C_VEL
LIN {X 0,Y 296.18,Z 592.56,A -85,B 0,C 180,E1 -16670.852,E2 -16670.852} C_VEL
LIN {X 0,Y 298.912,Z 584.45,A -85,B 0,C 180,E1 -16673.194,E2 -16673.194} C_VEL
LIN {X 0,Y 302.382,Z 574.93,A -85,B 0,C 180,E1 -16675.468,E2 -16675.468} C_VEL
LIN {X 0,Y 306.317,Z 563.81,A -85,B 0,C 180,E1 -16677.686,E2 -16677.686} C_VEL
LIN {X 0,Y 310.882,Z 550.777,A -85,B 0,C 180,E1 -16679.826,E2 -16679.826} C_VEL
LIN {X 0,Y 315.759,Z 536.5,A -85,B 0,C 180,E1 -16681.726,E2 -16681.726} C_VEL
LIN {X 0,Y 320.432,Z 522.225,A -85,B 0,C 180,E1 -16683.254,E2 -16683.254} C_VEL
LIN {X 0,Y 324.495,Z 508.626,A -85,B 0,C 180,E1 -16684.461,E2 -16684.461} C_VEL
LIN {X 0,Y 329.059,Z 492.246,A -85,B 0,C 180,E1 -16685.593,E2 -16685.593} C_VEL
LIN {X 0,Y 333.003,Z 475.731,A -85,B 0,C 180,E1 -16686.492,E2 -16686.492} C_VEL
LIN {X 0,Y 336.347,Z 458.143,A -85,B 0,C 180,E1 -16687.252,E2 -16687.252} C_VEL
LIN {X 0,Y 348.408,Z 391.823,A -85,B 0,C 180,E1 -16689.85,E2 -16689.85} C_VEL
LIN {X 0,Y 351.713,Z 375.142,A -85,B 0,C 180,E1 -16690.506,E2 -16690.506} C_VEL
LIN {X 0,Y 351.844,Z 373.325,A -85,B 0,C 180,E1 -16690.715,E2 -16690.715} C_VEL
LIN {X 0,Y 351.023,Z 368.347,A -85,B 0,C 180,E1 -16692.268,E2 -16692.268} C_VEL
LIN {X 0,Y 350.488,Z 364.318,A -85,B 0,C 180,E1 -16694.313,E2 -16694.313} C_VEL
LIN {X 0,Y 350.503,Z 363.102,A -85,B 0,C 180,E1 -16695.428,E2 -16695.428} C_VEL
LIN {X 0,Y 351.028,Z 363.226,A -85,B 0,C 180,E1 -16697.537,E2 -16697.537} C_VEL
LIN {X 0,Y 352.061,Z 364.346,A -85,B 0,C 180,E1 -16699.067,E2 -16699.067} C_VEL
LIN {X 0,Y 353.011,Z 366.055,A -85,B 0,C 180,E1 -16700.149,E2 -16700.149} C_VEL
LIN {X 0,Y 339.005,Z 437.778,A -85,B 0,C 180,E1 -16702.95,E2 -16702.95} C_VEL
LIN {X 0,Y 335.704,Z 456.158,A -85,B 0,C 180,E1 -16703.742,E2 -16703.742} C_VEL
LIN {X 0,Y 332.395,Z 471.708,A -85,B 0,C 180,E1 -16704.633,E2 -16704.633} C_VEL
LIN {X 0,Y 328.423,Z 487.664,A -85,B 0,C 180,E1 -16705.824,E2 -16705.824} C_VEL
LIN {X 0,Y 324.307,Z 502.22,A -85,B 0,C 180,E1 -16707.195,E2 -16707.195} C_VEL
LIN {X 0,Y 319.744,Z 516.713,A -85,B 0,C 180,E1 -16708.9,E2 -16708.9} C_VEL
LIN {X 0,Y 314.992,Z 530.465,A -85,B 0,C 180,E1 -16710.895,E2 -16710.895} C_VEL
LIN {X 0,Y 310.331,Z 542.733,A -85,B 0,C 180,E1 -16713.067,E2 -16713.067} C_VEL
LIN {X 0,Y 306.395,Z 552.7,A -85,B 0,C 180,E1 -16715.252,E2 -16715.252} C_VEL
LIN {X 0,Y 302.534,Z 562.206,A -85,B 0,C 180,E1 -16717.821,E2 -16717.821} C_VEL
LIN {X 0,Y 299.163,Z 569.903,A -85,B 0,C 180,E1 -16720.393,E2 -16720.393} C_VEL
LIN {X 0,Y 296.593,Z 575.592,A -85,B 0,C 180,E1 -16722.77,E2 -16722.77} C_VEL
LIN {X 0,Y 294.303,Z 580.635,A -85,B 0,C 180,E1 -16725.478,E2 -16725.478} C_VEL
LIN {X 0,Y 293.078,Z 583.542,A -85,B 0,C 180,E1 -16727.535,E2 -16727.535} C_VEL
LIN {X 0,Y 291.743,Z 586.366,A -85,B 0,C 180,E1 -16730.291,E2 -16730.291} C_VEL
LIN {X 0,Y 290.658,Z 587.973,A -85,B 0,C 180,E1 -16733.055,E2 -16733.055} C_VEL
LIN {X 0,Y 290.119,Z 588.345,A -85,B 0,C 180,E1 -16735.831,E2 -16735.831} C_VEL
LIN {X 0,Y 289.815,Z 587.512,A -85,B 0,C 180,E1 -16738.609,E2 -16738.609} C_VEL
LIN {X 0,Y 289.664,Z 585.451,A -85,B 0,C 180,E1 -16741.389,E2 -16741.389} C_VEL
LIN {X 0,Y 289.766,Z 582.101,A -85,B 0,C 180,E1 -16744.172,E2 -16744.172} C_VEL
LIN {X 0,Y 289.984,Z 577.158,A -85,B 0,C 180,E1 -16747.067,E2 -16747.067} C_VEL
LIN {X 0,Y 290.367,Z 571.139,A -85,B 0,C 180,E1 -16749.753,E2 -16749.753} C_VEL
LIN {X 0,Y 291.103,Z 563.226,A -85,B 0,C 180,E1 -16752.548,E2 -16752.548} C_VEL
LIN {X 0,Y 292.173,Z 554.734,A -85,B 0,C 180,E1 -16754.985,E2 -16754.985} C_VEL
LIN {X 0,Y 293.315,Z 544.461,A -85,B 0,C 180,E1 -16757.427,E2 -16757.427} C_VEL
LIN {X 0,Y 294.636,Z 533.97,A -85,B 0,C 180,E1 -16759.507,E2 -16759.507} C_VEL
LIN {X 0,Y 296.161,Z 522.657,A -85,B 0,C 180,E1 -16761.397,E2 -16761.397} C_VEL
LIN {X 0,Y 297.756,Z 509.563,A -85,B 0,C 180,E1 -16763.235,E2 -16763.235} C_VEL
LIN {X 0,Y 299.373,Z 495.993,A -85,B 0,C 180,E1 -16764.81,E2 -16764.81} C_VEL
LIN {X 0,Y 300.889,Z 481.816,A -85,B 0,C 180,E1 -16766.158,E2 -16766.158} C_VEL
LIN {X 0,Y 302.18,Z 467.592,A -85,B 0,C 180,E1 -16767.249,E2 -16767.249} C_VEL
LIN {X 0,Y 303.42,Z 451.455,A -85,B 0,C 180,E1 -16768.207,E2 -16768.207} C_VEL
LIN {X 0,Y 304.388,Z 435.368,A -85,B 0,C 180,E1 -16768.886,E2 -16768.886} C_VEL
LIN {X 0,Y 310.038,Z 330.005,A -85,B 0,C 180,E1 -16772.391,E2 -16772.391} C_VEL
LIN {X 0,Y 294.61,Z 294.711,A -85,B 0,C 180,E1 -16774.991,E2 -16774.991} C_VEL
LIN {X 0,Y 291.476,Z 287.455,A -85,B 0,C 180,E1 -16775.566,E2 -16775.566} C_VEL
LIN {X 0,Y 291.384,Z 286.815,A -85,B 0,C 180,E1 -16775.633,E2 -16775.633} C_VEL
LIN {X 0,Y 291.374,Z 286.816,A -85,B 0,C 180,E1 -16779.478,E2 -16779.478} C_VEL
LIN {X 0,Y 291.31,Z 286.825,A -85,B 0,C 180,E1 -16783.632,E2 -16783.632} C_VEL
LIN {X 0,Y 291.319,Z 286.822,A -85,B 0,C 180,E1 -16787.506,E2 -16787.506} C_VEL
LIN {X 0,Y 291.362,Z 286.814,A -85,B 0,C 180,E1 -16791.158,E2 -16791.158} C_VEL
LIN {X 0,Y 291.359,Z 286.814,A -85,B 0,C 180,E1 -16794.624,E2 -16794.624} C_VEL
LIN {X 0,Y 291.363,Z 286.817,A -85,B 0,C 180,E1 -16797.948,E2 -16797.948} C_VEL
LIN {X 0,Y 291.347,Z 286.817,A -85,B 0,C 180,E1 -16801.153,E2 -16801.153} C_VEL
LIN {X 0,Y 291.356,Z 286.816,A -85,B 0,C 180,E1 -16804.264,E2 -16804.264} C_VEL
LIN {X 0,Y 291.366,Z 286.815,A -85,B 0,C 180,E1 -16807.296,E2 -16807.296} C_VEL
LIN {X 0,Y 291.401,Z 286.81,A -85,B 0,C 180,E1 -16810.264,E2 -16810.264} C_VEL
LIN {X 0,Y 291.492,Z 286.798,A -85,B 0,C 180,E1 -16814.663,E2 -16814.663} C_VEL
LIN {X 0,Y 291.531,Z 286.793,A -85,B 0,C 180,E1 -16818.879,E2 -16818.879} C_VEL
LIN {X 0,Y 291.703,Z 286.776,A -85,B 0,C 180,E1 -16821.687,E2 -16821.687} C_VEL
LIN {X 0,Y 291.622,Z 286.781,A -85,B 0,C 180,E1 -16824.466,E2 -16824.466} C_VEL
LIN {X 0,Y 291.882,Z 286.749,A -85,B 0,C 180,E1 -16828.618,E2 -16828.618} C_VEL
LIN {X 0,Y 291.882,Z 286.752,A -85,B 0,C 180,E1 -16831.378,E2 -16831.378} C_VEL
LIN {X 0,Y 291.737,Z 286.768,A -85,B 0,C 180,E1 -16836.916,E2 -16836.916} C_VEL
LIN {X 0,Y 291.62,Z 286.784,A -85,B 0,C 180,E1 -16839.71,E2 -16839.71} C_VEL
LIN {X 0,Y 291.512,Z 286.797,A -85,B 0,C 180,E1 -16843.949,E2 -16843.949} C_VEL
LIN {X 0,Y 291.477,Z 286.8,A -85,B 0,C 180,E1 -16846.816,E2 -16846.816} C_VEL
LIN {X 0,Y 291.44,Z 286.805,A -85,B 0,C 180,E1 -16849.873,E2 -16849.873} C_VEL
LIN {X 0,Y 291.388,Z 286.811,A -85,B 0,C 180,E1 -16854.204,E2 -16854.204} C_VEL
LIN {X 0,Y 291.407,Z 286.812,A -85,B 0,C 180,E1 -16857.271,E2 -16857.271} C_VEL
LIN {X 0,Y 291.322,Z 286.819,A -85,B 0,C 180,E1 -16860.436,E2 -16860.436} C_VEL
LIN {X 0,Y 291.332,Z 286.819,A -85,B 0,C 180,E1 -16863.697,E2 -16863.697} C_VEL
LIN {X 0,Y 291.376,Z 286.816,A -85,B 0,C 180,E1 -16867.256,E2 -16867.256} C_VEL
LIN {X 0,Y 291.32,Z 286.82,A -85,B 0,C 180,E1 -16870.642,E2 -16870.642} C_VEL
LIN {X 0,Y 291.3,Z 286.821,A -85,B 0,C 180,E1 -16874.397,E2 -16874.397} C_VEL
LIN {X 0,Y 291.313,Z 286.82,A -85,B 0,C 180,E1 -16878.404,E2 -16878.404} C_VEL
LIN {X 0,Y 291.339,Z 286.821,A -85,B 0,C 180,E1 -16881.158,E2 -16881.158} C_VEL
LIN {X 0,Y 291.347,Z 286.816,A -85,B 0,C 180,E1 -16884.626,E2 -16884.626} C_VEL
LIN {X 0,Y 291.358,Z 286.815,A -85,B 0,C 180,E1 -16887.951,E2 -16887.951} C_VEL
LIN {X 0,Y 291.371,Z 286.817,A -85,B 0,C 180,E1 -16891.159,E2 -16891.159} C_VEL
LIN {X 0,Y 291.405,Z 286.808,A -85,B 0,C 180,E1 -16894.272,E2 -16894.272} C_VEL
LIN {X 0,Y 291.36,Z 286.817,A -85,B 0,C 180,E1 -16897.299,E2 -16897.299} C_VEL
LIN {X 0,Y 291.445,Z 286.803,A -85,B 0,C 180,E1 -16900.271,E2 -16900.271} C_VEL
LIN {X 0,Y 291.542,Z 286.793,A -85,B 0,C 180,E1 -16904.624,E2 -16904.624} C_VEL
LIN {X 0,Y 291.524,Z 286.796,A -85,B 0,C 180,E1 -16908.881,E2 -16908.881} C_VEL
LIN {X 0,Y 291.616,Z 286.782,A -85,B 0,C 180,E1 -16910.283,E2 -16910.283} C_VEL
LIN {X 0,Y 291.02,Z 286.862,A -85,B 0,C 180,E1 -16911.437,E2 -16911.437} C_VEL
LIN {X 0,Y 288.079,Z 287.227,A -85,B 0,C 180,E1 -16913.313,E2 -16913.313} C_VEL
LIN {X 0,Y 285.59,Z 287.536,A -85,B 0,C 180,E1 -16914.837,E2 -16914.837} C_VEL
LIN {X 0,Y 284.611,Z 287.655,A -85,B 0,C 180,E1 -16916.021,E2 -16916.021} C_VEL
LIN {X 0,Y 284.584,Z 287.658,A -85,B 0,C 180,E1 -16916.422,E2 -16916.422} C_VEL
LIN {X 0,Y 284.911,Z 287.617,A -85,B 0,C 180,E1 -16920.001,E2 -16920.001} C_VEL
LIN {X 0,Y 284.73,Z 287.643,A -85,B 0,C 180,E1 -16922.831,E2 -16922.831} C_VEL
LIN {X 0,Y 284.686,Z 287.65,A -85,B 0,C 180,E1 -16927.091,E2 -16927.091} C_VEL
LIN {X 0,Y 284.556,Z 287.661,A -85,B 0,C 180,E1 -16929.957,E2 -16929.957} C_VEL
LIN {X 0,Y 284.471,Z 287.673,A -85,B 0,C 180,E1 -16934.304,E2 -16934.304} C_VEL
LIN {X 0,Y 284.413,Z 287.683,A -85,B 0,C 180,E1 -16937.25,E2 -16937.25} C_VEL
LIN {X 0,Y 284.367,Z 287.687,A -85,B 0,C 180,E1 -16940.244,E2 -16940.244} C_VEL
LIN {X 0,Y 284.327,Z 287.696,A -85,B 0,C 180,E1 -16944.849,E2 -16944.849} C_VEL
LIN {X 0,Y 284.322,Z 287.692,A -85,B 0,C 180,E1 -16948.013,E2 -16948.013} C_VEL
LIN {X 0,Y 284.287,Z 287.697,A -85,B 0,C 180,E1 -16951.276,E2 -16951.276} C_VEL
LIN {X 0,Y 284.333,Z 287.691,A -85,B 0,C 180,E1 -16955.35,E2 -16955.35} C_VEL
LIN {X 0,Y 284.301,Z 287.694,A -85,B 0,C 180,E1 -16958.172,E2 -16958.172} C_VEL
LIN {X 0,Y 284.263,Z 287.698,A -85,B 0,C 180,E1 -16962.127,E2 -16962.127} C_VEL
LIN {X 0,Y 284.263,Z 287.699,A -85,B 0,C 180,E1 -16966.194,E2 -16966.194} C_VEL
LIN {X 0,Y 284.294,Z 287.704,A -85,B 0,C 180,E1 -16967.871,E2 -16967.871} C_VEL
LIN {X 0,Y 287.908,Z 302.294,A -85,B 0,C 180,E1 -16971.824,E2 -16971.824} C_VEL
LIN {X 0,Y 289.596,Z 309.344,A -85,B 0,C 180,E1 -16973.649,E2 -16973.649} C_VEL
LIN {X 0,Y 299.286,Z 335.602,A -85,B 0,C 180,E1 -16975.533,E2 -16975.533} C_VEL
LIN {X 0,Y 303.271,Z 366.044,A -85,B 0,C 180,E1 -16977.018,E2 -16977.018} C_VEL
LIN {X 0,Y 296.98,Z 477.086,A -85,B 0,C 180,E1 -16980.899,E2 -16980.899} C_VEL
LIN {X 0,Y 295.711,Z 492.397,A -85,B 0,C 180,E1 -16981.676,E2 -16981.676} C_VEL
LIN {X 0,Y 294.127,Z 507.673,A -85,B 0,C 180,E1 -16982.714,E2 -16982.714} C_VEL
LIN {X 0,Y 292.471,Z 522.341,A -85,B 0,C 180,E1 -16983.992,E2 -16983.992} C_VEL
LIN {X 0,Y 290.637,Z 536.637,A -85,B 0,C 180,E1 -16985.539,E2 -16985.539} C_VEL
LIN {X 0,Y 288.79,Z 550.468,A -85,B 0,C 180,E1 -16987.377,E2 -16987.377} C_VEL
LIN {X 0,Y 287.071,Z 563.02,A -85,B 0,C 180,E1 -16989.397,E2 -16989.397} C_VEL
LIN {X 0,Y 285.76,Z 573.224,A -85,B 0,C 180,E1 -16991.356,E2 -16991.356} C_VEL
LIN {X 0,Y 284.647,Z 582.708,A -85,B 0,C 180,E1 -16993.507,E2 -16993.507} C_VEL
LIN {X 0,Y 283.674,Z 591.947,A -85,B 0,C 180,E1 -16996.024,E2 -16996.024} C_VEL
LIN {X 0,Y 283.097,Z 599.563,A -85,B 0,C 180,E1 -16998.547,E2 -16998.547} C_VEL
LIN {X 0,Y 282.798,Z 606.497,A -85,B 0,C 180,E1 -17001.427,E2 -17001.427} C_VEL
LIN {X 0,Y 282.815,Z 611.77,A -85,B 0,C 180,E1 -17004.297,E2 -17004.297} C_VEL
LIN {X 0,Y 282.668,Z 615.462,A -85,B 0,C 180,E1 -17007.152,E2 -17007.152} C_VEL
LIN {X 0,Y 282.883,Z 616.797,A -85,B 0,C 180,E1 -17008.578,E2 -17008.578} C_VEL
LIN {X 0,Y 282.885,Z 617.76,A -85,B 0,C 180,E1 -17010.002,E2 -17010.002} C_VEL
LIN {X 0,Y 282.517,Z 618.652,A -85,B 0,C 180,E1 -17012.854,E2 -17012.854} C_VEL
LIN {X 0,Y 282.484,Z 618.235,A -85,B 0,C 180,E1 -17015.713,E2 -17015.713} C_VEL
LIN {X 0,Y 282.528,Z 616.532,A -85,B 0,C 180,E1 -17018.585,E2 -17018.585} C_VEL
LIN {X 0,Y 283.001,Z 613.619,A -85,B 0,C 180,E1 -17021.461,E2 -17021.461} C_VEL
LIN {X 0,Y 284.072,Z 609.48,A -85,B 0,C 180,E1 -17024.326,E2 -17024.326} C_VEL
LIN {X 0,Y 285.777,Z 604.055,A -85,B 0,C 180,E1 -17027.166,E2 -17027.166} C_VEL
LIN {X 0,Y 288.182,Z 597.255,A -85,B 0,C 180,E1 -17029.965,E2 -17029.965} C_VEL
LIN {X 0,Y 291.116,Z 589.002,A -85,B 0,C 180,E1 -17032.724,E2 -17032.724} C_VEL
LIN {X 0,Y 295.05,Z 579.06,A -85,B 0,C 180,E1 -17035.39,E2 -17035.39} C_VEL
LIN {X 0,Y 299.028,Z 568.851,A -85,B 0,C 180,E1 -17037.659,E2 -17037.659} C_VEL
LIN {X 0,Y 303.595,Z 556.929,A -85,B 0,C 180,E1 -17039.85,E2 -17039.85} C_VEL
LIN {X 0,Y 308.482,Z 544.018,A -85,B 0,C 180,E1 -17041.794,E2 -17041.794} C_VEL
LIN {X 0,Y 313.053,Z 531.375,A -85,B 0,C 180,E1 -17043.37,E2 -17043.37} C_VEL
LIN {X 0,Y 318.582,Z 515.059,A -85,B 0,C 180,E1 -17045.001,E2 -17045.001} C_VEL
LIN {X 0,Y 323.163,Z 500.451,A -85,B 0,C 180,E1 -17046.152,E2 -17046.152} C_VEL
LIN {X 0,Y 327.749,Z 484.001,A -85,B 0,C 180,E1 -17047.175,E2 -17047.175} C_VEL
LIN {X 0,Y 332.094,Z 465.028,A -85,B 0,C 180,E1 -17048.101,E2 -17048.101} C_VEL
LIN {X 0,Y 346.187,Z 393.064,A -85,B 0,C 180,E1 -17050.94,E2 -17050.94} C_VEL
LIN {X 0,Y 349.349,Z 378.086,A -85,B 0,C 180,E1 -17051.527,E2 -17051.527} C_VEL
LIN {X 0,Y 348.85,Z 374.159,A -85,B 0,C 180,E1 -17052.894,E2 -17052.894} C_VEL
LIN {X 0,Y 348.632,Z 370.691,A -85,B 0,C 180,E1 -17054.788,E2 -17054.788} C_VEL
LIN {X 0,Y 348.709,Z 369.935,A -85,B 0,C 180,E1 -17055.554,E2 -17055.554} C_VEL
LIN {X 0,Y 349.258,Z 370.12,A -85,B 0,C 180,E1 -17057.609,E2 -17057.609} C_VEL
LIN {X 0,Y 350.104,Z 371.137,A -85,B 0,C 180,E1 -17058.932,E2 -17058.932} C_VEL
LIN {X 0,Y 350.301,Z 371.529,A -85,B 0,C 180,E1 -17059.198,E2 -17059.198} C_VEL
LIN {X 0,Y 335.622,Z 442.245,A -85,B 0,C 180,E1 -17061.991,E2 -17061.991} C_VEL
LIN {X 0,Y 332.195,Z 459.556,A -85,B 0,C 180,E1 -17062.775,E2 -17062.775} C_VEL
LIN {X 0,Y 328.849,Z 473.787,A -85,B 0,C 180,E1 -17063.625,E2 -17063.625} C_VEL
LIN {X 0,Y 324.67,Z 489.214,A -85,B 0,C 180,E1 -17064.806,E2 -17064.806} C_VEL
LIN {X 0,Y 320.302,Z 503.417,A -85,B 0,C 180,E1 -17066.166,E2 -17066.166} C_VEL
LIN {X 0,Y 315.203,Z 518.278,A -85,B 0,C 180,E1 -17067.953,E2 -17067.953} C_VEL
LIN {X 0,Y 310.603,Z 530.544,A -85,B 0,C 180,E1 -17069.761,E2 -17069.761} C_VEL
LIN {X 0,Y 305.751,Z 542.477,A -85,B 0,C 180,E1 -17071.886,E2 -17071.886} C_VEL
LIN {X 0,Y 301.427,Z 552.508,A -85,B 0,C 180,E1 -17074.076,E2 -17074.076} C_VEL
LIN {X 0,Y 297.216,Z 562.062,A -85,B 0,C 180,E1 -17076.666,E2 -17076.666} C_VEL
LIN {X 0,Y 293.978,Z 569.011,A -85,B 0,C 180,E1 -17078.985,E2 -17078.985} C_VEL
LIN {X 0,Y 290.629,Z 575.599,A -85,B 0,C 180,E1 -17081.676,E2 -17081.676} C_VEL
LIN {X 0,Y 288.152,Z 580.723,A -85,B 0,C 180,E1 -17084.437,E2 -17084.437} C_VEL
LIN {X 0,Y 286.996,Z 582.822,A -85,B 0,C 180,E1 -17085.824,E2 -17085.824} C_VEL
LIN {X 0,Y 285.498,Z 586.01,A -85,B 0,C 180,E1 -17088.641,E2 -17088.641} C_VEL
LIN {X 0,Y 284.142,Z 588.047,A -85,B 0,C 180,E1 -17091.464,E2 -17091.464} C_VEL
LIN {X 0,Y 283.259,Z 588.892,A -85,B 0,C 180,E1 -17094.303,E2 -17094.303} C_VEL
LIN {X 0,Y 282.912,Z 588.49,A -85,B 0,C 180,E1 -17097.151,E2 -17097.151} C_VEL
LIN {X 0,Y 282.596,Z 586.87,A -85,B 0,C 180,E1 -17099.999,E2 -17099.999} C_VEL
LIN {X 0,Y 282.631,Z 583.993,A -85,B 0,C 180,E1 -17102.849,E2 -17102.849} C_VEL
LIN {X 0,Y 282.722,Z 579.782,A -85,B 0,C 180,E1 -17105.705,E2 -17105.705} C_VEL
LIN {X 0,Y 283.084,Z 574.13,A -85,B 0,C 180,E1 -17108.565,E2 -17108.565} C_VEL
LIN {X 0,Y 283.629,Z 566.874,A -85,B 0,C 180,E1 -17111.432,E2 -17111.432} C_VEL
LIN {X 0,Y 284.614,Z 559.031,A -85,B 0,C 180,E1 -17113.93,E2 -17113.93} C_VEL
LIN {X 0,Y 285.555,Z 550.159,A -85,B 0,C 180,E1 -17116.285,E2 -17116.285} C_VEL
LIN {X 0,Y 286.878,Z 539.881,A -85,B 0,C 180,E1 -17118.569,E2 -17118.569} C_VEL
LIN {X 0,Y 288.427,Z 528.492,A -85,B 0,C 180,E1 -17120.689,E2 -17120.689} C_VEL
LIN {X 0,Y 289.954,Z 516.072,A -85,B 0,C 180,E1 -17122.629,E2 -17122.629} C_VEL
LIN {X 0,Y 291.714,Z 502.675,A -85,B 0,C 180,E1 -17124.365,E2 -17124.365} C_VEL
LIN {X 0,Y 293.376,Z 488.049,A -85,B 0,C 180,E1 -17125.923,E2 -17125.923} C_VEL
LIN {X 0,Y 294.965,Z 473.034,A -85,B 0,C 180,E1 -17127.203,E2 -17127.203} C_VEL
LIN {X 0,Y 296.221,Z 456.913,A -85,B 0,C 180,E1 -17128.278,E2 -17128.278} C_VEL
LIN {X 0,Y 297.35,Z 440.673,A -85,B 0,C 180,E1 -17129.063,E2 -17129.063} C_VEL
LIN {X 0,Y 303.387,Z 331.847,A -85,B 0,C 180,E1 -17132.822,E2 -17132.822} C_VEL
LIN {X 0,Y 288.566,Z 297.908,A -85,B 0,C 180,E1 -17135.388,E2 -17135.388} C_VEL
LIN {X 0,Y 284.411,Z 288.108,A -85,B 0,C 180,E1 -17136.166,E2 -17136.166} C_VEL
LIN {X 0,Y 284.351,Z 287.691,A -85,B 0,C 180,E1 -17136.221,E2 -17136.221} C_VEL
LIN {X 0,Y 284.306,Z 287.698,A -85,B 0,C 180,E1 -17139.993,E2 -17139.993} C_VEL
LIN {X 0,Y 284.246,Z 287.703,A -85,B 0,C 180,E1 -17144.188,E2 -17144.188} C_VEL
LIN {X 0,Y 284.271,Z 287.7,A -85,B 0,C 180,E1 -17148.122,E2 -17148.122} C_VEL
LIN {X 0,Y 284.326,Z 287.692,A -85,B 0,C 180,E1 -17152.275,E2 -17152.275} C_VEL
LIN {X 0,Y 284.307,Z 287.694,A -85,B 0,C 180,E1 -17155.349,E2 -17155.349} C_VEL
LIN {X 0,Y 284.283,Z 287.695,A -85,B 0,C 180,E1 -17158.722,E2 -17158.722} C_VEL
LIN {X 0,Y 284.284,Z 287.699,A -85,B 0,C 180,E1 -17161.982,E2 -17161.982} C_VEL
LIN {X 0,Y 284.318,Z 287.693,A -85,B 0,C 180,E1 -17166.144,E2 -17166.144} C_VEL
LIN {X 0,Y 284.372,Z 287.688,A -85,B 0,C 180,E1 -17169.902,E2 -17169.902} C_VEL
LIN {X 0,Y 284.441,Z 287.677,A -85,B 0,C 180,E1 -17174.491,E2 -17174.491} C_VEL
LIN {X 0,Y 284.482,Z 287.671,A -85,B 0,C 180,E1 -17178.599,E2 -17178.599} C_VEL
LIN {X 0,Y 284.653,Z 287.654,A -85,B 0,C 180,E1 -17181.479,E2 -17181.479} C_VEL
LIN {X 0,Y 284.593,Z 287.657,A -85,B 0,C 180,E1 -17184.329,E2 -17184.329} C_VEL
LIN {X 0,Y 284.848,Z 287.626,A -85,B 0,C 180,E1 -17188.584,E2 -17188.584} C_VEL
LIN {X 0,Y 284.848,Z 287.629,A -85,B 0,C 180,E1 -17191.412,E2 -17191.412} C_VEL
LIN {X 0,Y 284.689,Z 287.647,A -85,B 0,C 180,E1 -17197.088,E2 -17197.088} C_VEL
LIN {X 0,Y 284.557,Z 287.662,A -85,B 0,C 180,E1 -17199.954,E2 -17199.954} C_VEL
LIN {X 0,Y 284.472,Z 287.672,A -85,B 0,C 180,E1 -17204.301,E2 -17204.301} C_VEL
LIN {X 0,Y 284.415,Z 287.682,A -85,B 0,C 180,E1 -17207.247,E2 -17207.247} C_VEL
LIN {X 0,Y 284.368,Z 287.685,A -85,B 0,C 180,E1 -17210.241,E2 -17210.241} C_VEL
LIN {X 0,Y 284.358,Z 287.688,A -85,B 0,C 180,E1 -17213.874,E2 -17213.874} C_VEL
LIN {X 0,Y 284.382,Z 287.685,A -85,B 0,C 180,E1 -17217.171,E2 -17217.171} C_VEL
LIN {X 0,Y 284.281,Z 287.7,A -85,B 0,C 180,E1 -17221.273,E2 -17221.273} C_VEL
LIN {X 0,Y 284.349,Z 287.691,A -85,B 0,C 180,E1 -17225.353,E2 -17225.353} C_VEL
LIN {X 0,Y 284.304,Z 287.693,A -85,B 0,C 180,E1 -17228.167,E2 -17228.167} C_VEL
LIN {X 0,Y 284.256,Z 287.699,A -85,B 0,C 180,E1 -17232.124,E2 -17232.124} C_VEL
LIN {X 0,Y 284.255,Z 287.699,A -85,B 0,C 180,E1 -17236.191,E2 -17236.191} C_VEL
LIN {X 0,Y 284.293,Z 287.694,A -85,B 0,C 180,E1 -17240.023,E2 -17240.023} C_VEL
LIN {X 0,Y 284.318,Z 287.693,A -85,B 0,C 180,E1 -17243.614,E2 -17243.614} C_VEL
LIN {X 0,Y 284.294,Z 287.699,A -85,B 0,C 180,E1 -17247.189,E2 -17247.189} C_VEL
LIN {X 0,Y 284.345,Z 287.687,A -85,B 0,C 180,E1 -17250.376,E2 -17250.376} C_VEL
LIN {X 0,Y 284.366,Z 287.687,A -85,B 0,C 180,E1 -17253.587,E2 -17253.587} C_VEL
LIN {X 0,Y 284.319,Z 287.693,A -85,B 0,C 180,E1 -17256.704,E2 -17256.704} C_VEL
LIN {X 0,Y 284.386,Z 287.687,A -85,B 0,C 180,E1 -17261.262,E2 -17261.262} C_VEL
LIN {X 0,Y 284.479,Z 287.672,A -85,B 0,C 180,E1 -17264.46,E2 -17264.46} C_VEL
LIN {X 0,Y 284.475,Z 287.672,A -85,B 0,C 180,E1 -17268.602,E2 -17268.602} C_VEL
LIN {X 0,Y 284.644,Z 287.653,A -85,B 0,C 180,E1 -17271.482,E2 -17271.482} C_VEL
LIN {X 0,Y 284.585,Z 287.658,A -85,B 0,C 180,E1 -17274.332,E2 -17274.332} C_VEL
LIN {X 0,Y 284.584,Z 287.658,A -85,B 0,C 180,E1 -17276.422,E2 -17276.422} C_VEL
LIN {X 0,Y 284.069,Z 287.725,A -85,B 0,C 180,E1 -17277.605,E2 -17277.605} C_VEL
LIN {X 0,Y 282.569,Z 287.912,A -85,B 0,C 180,E1 -17278.768,E2 -17278.768} C_VEL
LIN {X 0,Y 278.866,Z 288.375,A -85,B 0,C 180,E1 -17281.102,E2 -17281.102} C_VEL
LIN {X 0,Y 277.789,Z 288.506,A -85,B 0,C 180,E1 -17282.316,E2 -17282.316} C_VEL
LIN {X 0,Y 277.691,Z 288.519,A -85,B 0,C 180,E1 -17282.728,E2 -17282.728} C_VEL
LIN {X 0,Y 277.641,Z 288.526,A -85,B 0,C 180,E1 -17287.272,E2 -17287.272} C_VEL
LIN {X 0,Y 277.496,Z 288.541,A -85,B 0,C 180,E1 -17290.213,E2 -17290.213} C_VEL
LIN {X 0,Y 277.424,Z 288.553,A -85,B 0,C 180,E1 -17294.676,E2 -17294.676} C_VEL
LIN {X 0,Y 277.333,Z 288.565,A -85,B 0,C 180,E1 -17299.236,E2 -17299.236} C_VEL
LIN {X 0,Y 277.282,Z 288.569,A -85,B 0,C 180,E1 -17304.159,E2 -17304.159} C_VEL
LIN {X 0,Y 277.316,Z 288.565,A -85,B 0,C 180,E1 -17307.506,E2 -17307.506} C_VEL
LIN {X 0,Y 277.264,Z 288.573,A -85,B 0,C 180,E1 -17310.483,E2 -17310.483} C_VEL
LIN {X 0,Y 277.239,Z 288.574,A -85,B 0,C 180,E1 -17313.898,E2 -17313.898} C_VEL
LIN {X 0,Y 277.257,Z 288.572,A -85,B 0,C 180,E1 -17317.472,E2 -17317.472} C_VEL
LIN {X 0,Y 277.203,Z 288.578,A -85,B 0,C 180,E1 -17321.239,E2 -17321.239} C_VEL
LIN {X 0,Y 277.211,Z 288.578,A -85,B 0,C 180,E1 -17325.225,E2 -17325.225} C_VEL
LIN {X 0,Y 277.251,Z 288.609,A -85,B 0,C 180,E1 -17327.385,E2 -17327.385} C_VEL
LIN {X 0,Y 280.857,Z 303.214,A -85,B 0,C 180,E1 -17331.442,E2 -17331.442} C_VEL
LIN {X 0,Y 282.335,Z 309.315,A -85,B 0,C 180,E1 -17333.006,E2 -17333.006} C_VEL
LIN {X 0,Y 292.863,Z 337.736,A -85,B 0,C 180,E1 -17335.102,E2 -17335.102} C_VEL
LIN {X 0,Y 296.581,Z 366.928,A -85,B 0,C 180,E1 -17336.563,E2 -17336.563} C_VEL
LIN {X 0,Y 290.167,Z 476.785,A -85,B 0,C 180,E1 -17340.532,E2 -17340.532} C_VEL
LIN {X 0,Y 288.748,Z 493.318,A -85,B 0,C 180,E1 -17341.408,E2 -17341.408} C_VEL
LIN {X 0,Y 286.983,Z 509.487,A -85,B 0,C 180,E1 -17342.57,E2 -17342.57} C_VEL
LIN {X 0,Y 285.327,Z 523.706,A -85,B 0,C 180,E1 -17343.88,E2 -17343.88} C_VEL
LIN {X 0,Y 283.51,Z 537.685,A -85,B 0,C 180,E1 -17345.469,E2 -17345.469} C_VEL
LIN {X 0,Y 281.769,Z 550.205,A -85,B 0,C 180,E1 -17347.193,E2 -17347.193} C_VEL
LIN {X 0,Y 280.045,Z 562.596,A -85,B 0,C 180,E1 -17349.241,E2 -17349.241} C_VEL
LIN {X 0,Y 278.529,Z 574.509,A -85,B 0,C 180,E1 -17351.617,E2 -17351.617} C_VEL
LIN {X 0,Y 277.436,Z 583.714,A -85,B 0,C 180,E1 -17353.822,E2 -17353.822} C_VEL
LIN {X 0,Y 276.509,Z 592.717,A -85,B 0,C 180,E1 -17356.404,E2 -17356.404} C_VEL
LIN {X 0,Y 275.946,Z 600.091,A -85,B 0,C 180,E1 -17358.99,E2 -17358.99} C_VEL
LIN {X 0,Y 275.726,Z 606.807,A -85,B 0,C 180,E1 -17361.943,E2 -17361.943} C_VEL
LIN {X 0,Y 275.733,Z 610.762,A -85,B 0,C 180,E1 -17364.15,E2 -17364.15} C_VEL
LIN {X 0,Y 275.599,Z 614.635,A -85,B 0,C 180,E1 -17367.079,E2 -17367.079} C_VEL
LIN {X 0,Y 275.825,Z 616.052,A -85,B 0,C 180,E1 -17368.542,E2 -17368.542} C_VEL
LIN {X 0,Y 275.832,Z 617.089,A -85,B 0,C 180,E1 -17370.002,E2 -17370.002} C_VEL
LIN {X 0,Y 275.441,Z 618.089,A -85,B 0,C 180,E1 -17372.927,E2 -17372.927} C_VEL
LIN {X 0,Y 275.389,Z 617.812,A -85,B 0,C 180,E1 -17375.861,E2 -17375.861} C_VEL
LIN {X 0,Y 275.448,Z 616.29,A -85,B 0,C 180,E1 -17378.808,E2 -17378.808} C_VEL
LIN {X 0,Y 275.983,Z 613.571,A -85,B 0,C 180,E1 -17381.757,E2 -17381.757} C_VEL
LIN {X 0,Y 277.147,Z 609.641,A -85,B 0,C 180,E1 -17384.692,E2 -17384.692} C_VEL
LIN {X 0,Y 278.958,Z 604.416,A -85,B 0,C 180,E1 -17387.599,E2 -17387.599} C_VEL
LIN {X 0,Y 281.52,Z 597.853,A -85,B 0,C 180,E1 -17390.459,E2 -17390.459} C_VEL
LIN {X 0,Y 284.625,Z 589.909,A -85,B 0,C 180,E1 -17393.272,E2 -17393.272} C_VEL
LIN {X 0,Y 288.769,Z 580.363,A -85,B 0,C 180,E1 -17395.983,E2 -17395.983} C_VEL
LIN {X 0,Y 292.94,Z 570.55,A -85,B 0,C 180,E1 -17398.285,E2 -17398.285} C_VEL
LIN {X 0,Y 297.713,Z 559.171,A -85,B 0,C 180,E1 -17400.502,E2 -17400.502} C_VEL
LIN {X 0,Y 303.179,Z 545.912,A -85,B 0,C 180,E1 -17402.615,E2 -17402.615} C_VEL
LIN {X 0,Y 308.417,Z 532.623,A -85,B 0,C 180,E1 -17404.334,E2 -17404.334} C_VEL
LIN {X 0,Y 314.223,Z 517.005,A -85,B 0,C 180,E1 -17405.954,E2 -17405.954} C_VEL
LIN {X 0,Y 318.981,Z 503.141,A -85,B 0,C 180,E1 -17407.097,E2 -17407.097} C_VEL
LIN {X 0,Y 324.332,Z 485.514,A -85,B 0,C 180,E1 -17408.239,E2 -17408.239} C_VEL
LIN {X 0,Y 329.31,Z 465.884,A -85,B 0,C 180,E1 -17409.218,E2 -17409.218} C_VEL
LIN {X 0,Y 345.778,Z 387.886,A -85,B 0,C 180,E1 -17412.301,E2 -17412.301} C_VEL
LIN {X 0,Y 346.952,Z 382.604,A -85,B 0,C 180,E1 -17412.522,E2 -17412.522} C_VEL
LIN {X 0,Y 346.772,Z 379.96,A -85,B 0,C 180,E1 -17413.559,E2 -17413.559} C_VEL
LIN {X 0,Y 346.826,Z 377.181,A -85,B 0,C 180,E1 -17415.174,E2 -17415.174} C_VEL
LIN {X 0,Y 346.907,Z 376.735,A -85,B 0,C 180,E1 -17415.858,E2 -17415.858} C_VEL
LIN {X 0,Y 347.596,Z 377.136,A -85,B 0,C 180,E1 -17417.91,E2 -17417.91} C_VEL
LIN {X 0,Y 347.796,Z 377.364,A -85,B 0,C 180,E1 -17418.254,E2 -17418.254} C_VEL
LIN {X 0,Y 330.762,Z 455.248,A -85,B 0,C 180,E1 -17421.379,E2 -17421.379} C_VEL
LIN {X 0,Y 327.041,Z 470.735,A -85,B 0,C 180,E1 -17422.232,E2 -17422.232} C_VEL
LIN {X 0,Y 323.045,Z 484.932,A -85,B 0,C 180,E1 -17423.253,E2 -17423.253} C_VEL
LIN {X 0,Y 318.271,Z 499.692,A -85,B 0,C 180,E1 -17424.573,E2 -17424.573} C_VEL
LIN {X 0,Y 313.04,Z 514.354,A -85,B 0,C 180,E1 -17426.243,E2 -17426.243} C_VEL
LIN {X 0,Y 308.828,Z 525.066,A -85,B 0,C 180,E1 -17427.7,E2 -17427.7} C_VEL
LIN {X 0,Y 303.565,Z 537.583,A -85,B 0,C 180,E1 -17429.764,E2 -17429.764} C_VEL
LIN {X 0,Y 298.61,Z 548.381,A -85,B 0,C 180,E1 -17431.918,E2 -17431.918} C_VEL
LIN {X 0,Y 294.272,Z 557.484,A -85,B 0,C 180,E1 -17434.159,E2 -17434.159} C_VEL
LIN {X 0,Y 289.983,Z 566.196,A -85,B 0,C 180,E1 -17436.806,E2 -17436.806} C_VEL
LIN {X 0,Y 286.627,Z 572.543,A -85,B 0,C 180,E1 -17439.173,E2 -17439.173} C_VEL
LIN {X 0,Y 283.337,Z 578.468,A -85,B 0,C 180,E1 -17441.936,E2 -17441.936} C_VEL
LIN {X 0,Y 281.441,Z 582.013,A -85,B 0,C 180,E1 -17444.056,E2 -17444.056} C_VEL
LIN {X 0,Y 280.204,Z 583.989,A -85,B 0,C 180,E1 -17445.473,E2 -17445.473} C_VEL
LIN {X 0,Y 278.593,Z 586.944,A -85,B 0,C 180,E1 -17448.356,E2 -17448.356} C_VEL
LIN {X 0,Y 276.932,Z 588.999,A -85,B 0,C 180,E1 -17451.798,E2 -17451.798} C_VEL
LIN {X 0,Y 276.227,Z 589.408,A -85,B 0,C 180,E1 -17454.158,E2 -17454.158} C_VEL
LIN {X 0,Y 275.829,Z 588.849,A -85,B 0,C 180,E1 -17457.078,E2 -17457.078} C_VEL
LIN {X 0,Y 275.508,Z 587.081,A -85,B 0,C 180,E1 -17459.999,E2 -17459.999} C_VEL
LIN {X 0,Y 275.556,Z 584.025,A -85,B 0,C 180,E1 -17462.923,E2 -17462.923} C_VEL
LIN {X 0,Y 275.644,Z 579.62,A -85,B 0,C 180,E1 -17465.852,E2 -17465.852} C_VEL
LIN {X 0,Y 276.02,Z 573.769,A -85,B 0,C 180,E1 -17468.786,E2 -17468.786} C_VEL
LIN {X 0,Y 276.525,Z 567.291,A -85,B 0,C 180,E1 -17471.359,E2 -17471.359} C_VEL
LIN {X 0,Y 277.494,Z 559.434,A -85,B 0,C 180,E1 -17473.921,E2 -17473.921} C_VEL
LIN {X 0,Y 278.558,Z 549.846,A -85,B 0,C 180,E1 -17476.512,E2 -17476.512} C_VEL
LIN {X 0,Y 279.809,Z 540.271,A -85,B 0,C 180,E1 -17478.676,E2 -17478.676} C_VEL
LIN {X 0,Y 281.366,Z 528.876,A -85,B 0,C 180,E1 -17480.85,E2 -17480.85} C_VEL
LIN {X 0,Y 282.961,Z 516.447,A -85,B 0,C 180,E1 -17482.834,E2 -17482.834} C_VEL
LIN {X 0,Y 284.715,Z 503.172,A -85,B 0,C 180,E1 -17484.596,E2 -17484.596} C_VEL
LIN {X 0,Y 286.437,Z 488.417,A -85,B 0,C 180,E1 -17486.207,E2 -17486.207} C_VEL
LIN {X 0,Y 288.065,Z 473.457,A -85,B 0,C 180,E1 -17487.516,E2 -17487.516} C_VEL
LIN {X 0,Y 289.297,Z 458.208,A -85,B 0,C 180,E1 -17488.571,E2 -17488.571} C_VEL
LIN {X 0,Y 290.455,Z 442.034,A -85,B 0,C 180,E1 -17489.396,E2 -17489.396} C_VEL
LIN {X 0,Y 296.747,Z 333.785,A -85,B 0,C 180,E1 -17493.252,E2 -17493.252} C_VEL
LIN {X 0,Y 282.675,Z 301.397,A -85,B 0,C 180,E1 -17495.758,E2 -17495.758} C_VEL
LIN {X 0,Y 277.367,Z 289.1,A -85,B 0,C 180,E1 -17496.781,E2 -17496.781} C_VEL
LIN {X 0,Y 277.295,Z 288.568,A -85,B 0,C 180,E1 -17496.857,E2 -17496.857} C_VEL
LIN {X 0,Y 277.21,Z 288.58,A -85,B 0,C 180,E1 -17501.235,E2 -17501.235} C_VEL
LIN {X 0,Y 277.201,Z 288.58,A -85,B 0,C 180,E1 -17505.224,E2 -17505.224} C_VEL
LIN {X 0,Y 277.222,Z 288.578,A -85,B 0,C 180,E1 -17509.51,E2 -17509.51} C_VEL
LIN {X 0,Y 277.27,Z 288.57,A -85,B 0,C 180,E1 -17512.529,E2 -17512.529} C_VEL
LIN {X 0,Y 277.245,Z 288.576,A -85,B 0,C 180,E1 -17516.102,E2 -17516.102} C_VEL
LIN {X 0,Y 277.259,Z 288.573,A -85,B 0,C 180,E1 -17519.536,E2 -17519.536} C_VEL
LIN {X 0,Y 277.291,Z 288.567,A -85,B 0,C 180,E1 -17522.855,E2 -17522.855} C_VEL
LIN {X 0,Y 277.279,Z 288.57,A -85,B 0,C 180,E1 -17526.073,E2 -17526.073} C_VEL
LIN {X 0,Y 277.3,Z 288.566,A -85,B 0,C 180,E1 -17530.761,E2 -17530.761} C_VEL
LIN {X 0,Y 277.404,Z 288.556,A -85,B 0,C 180,E1 -17535.322,E2 -17535.322} C_VEL
LIN {X 0,Y 277.501,Z 288.545,A -85,B 0,C 180,E1 -17539.787,E2 -17539.787} C_VEL
LIN {X 0,Y 277.646,Z 288.523,A -85,B 0,C 180,E1 -17542.727,E2 -17542.727} C_VEL
LIN {X 0,Y 277.814,Z 288.502,A -85,B 0,C 180,E1 -17548.548,E2 -17548.548} C_VEL
LIN {X 0,Y 277.813,Z 288.505,A -85,B 0,C 180,E1 -17551.448,E2 -17551.448} C_VEL
LIN {X 0,Y 277.644,Z 288.526,A -85,B 0,C 180,E1 -17557.269,E2 -17557.269} C_VEL
LIN {X 0,Y 277.498,Z 288.54,A -85,B 0,C 180,E1 -17560.209,E2 -17560.209} C_VEL
LIN {X 0,Y 277.425,Z 288.55,A -85,B 0,C 180,E1 -17564.672,E2 -17564.672} C_VEL
LIN {X 0,Y 277.334,Z 288.563,A -85,B 0,C 180,E1 -17569.232,E2 -17569.232} C_VEL
LIN {X 0,Y 277.307,Z 288.565,A -85,B 0,C 180,E1 -17574.169,E2 -17574.169} C_VEL
LIN {X 0,Y 277.311,Z 288.568,A -85,B 0,C 180,E1 -17577.503,E2 -17577.503} C_VEL
LIN {X 0,Y 277.26,Z 288.571,A -85,B 0,C 180,E1 -17580.48,E2 -17580.48} C_VEL
LIN {X 0,Y 277.242,Z 288.573,A -85,B 0,C 180,E1 -17583.894,E2 -17583.894} C_VEL
LIN {X 0,Y 277.264,Z 288.574,A -85,B 0,C 180,E1 -17587.467,E2 -17587.467} C_VEL
LIN {X 0,Y 277.197,Z 288.583,A -85,B 0,C 180,E1 -17591.236,E2 -17591.236} C_VEL
LIN {X 0,Y 277.203,Z 288.581,A -85,B 0,C 180,E1 -17595.223,E2 -17595.223} C_VEL
LIN {X 0,Y 277.209,Z 288.579,A -85,B 0,C 180,E1 -17599.512,E2 -17599.512} C_VEL
LIN {X 0,Y 277.254,Z 288.57,A -85,B 0,C 180,E1 -17602.53,E2 -17602.53} C_VEL
LIN {X 0,Y 277.233,Z 288.574,A -85,B 0,C 180,E1 -17606.104,E2 -17606.104} C_VEL
LIN {X 0,Y 277.248,Z 288.573,A -85,B 0,C 180,E1 -17609.539,E2 -17609.539} C_VEL
LIN {X 0,Y 277.347,Z 288.561,A -85,B 0,C 180,E1 -17612.864,E2 -17612.864} C_VEL
LIN {X 0,Y 277.284,Z 288.568,A -85,B 0,C 180,E1 -17616.077,E2 -17616.077} C_VEL
LIN {X 0,Y 277.329,Z 288.563,A -85,B 0,C 180,E1 -17620.766,E2 -17620.766} C_VEL
LIN {X 0,Y 277.421,Z 288.553,A -85,B 0,C 180,E1 -17625.326,E2 -17625.326} C_VEL
LIN {X 0,Y 277.494,Z 288.542,A -85,B 0,C 180,E1 -17629.789,E2 -17629.789} C_VEL
LIN {X 0,Y 277.636,Z 288.526,A -85,B 0,C 180,E1 -17632.73,E2 -17632.73} C_VEL
LIN {X 0,Y 277.809,Z 288.503,A -85,B 0,C 180,E1 -17638.552,E2 -17638.552} C_VEL
LIN {X 0,Y 277.81,Z 288.503,A -85,B 0,C 180,E1 -17641.451,E2 -17641.451} C_VEL
LIN {X 0,Y 277.691,Z 288.519,A -85,B 0,C 180,E1 -17642.728,E2 -17642.728} C_VEL
LIN {X 0,Y 276.99,Z 288.615,A -85,B 0,C 180,E1 -17643.937,E2 -17643.937} C_VEL
LIN {X 0,Y 274.1,Z 288.981,A -85,B 0,C 180,E1 -17645.906,E2 -17645.906} C_VEL
LIN {X 0,Y 271.673,Z 289.28,A -85,B 0,C 180,E1 -17647.507,E2 -17647.507} C_VEL
LIN {X 0,Y 270.644,Z 289.401,A -85,B 0,C 180,E1 -17648.747,E2 -17648.747} C_VEL
LIN {X 0,Y 270.566,Z 289.407,A -85,B 0,C 180,E1 -17649.168,E2 -17649.168} C_VEL
LIN {X 0,Y 270.349,Z 289.433,A -85,B 0,C 180,E1 -17653.532,E2 -17653.532} C_VEL
LIN {X 0,Y 270.344,Z 289.435,A -85,B 0,C 180,E1 -17656.617,E2 -17656.617} C_VEL
LIN {X 0,Y 270.282,Z 289.444,A -85,B 0,C 180,E1 -17660.603,E2 -17660.603} C_VEL
LIN {X 0,Y 270.228,Z 289.45,A -85,B 0,C 180,E1 -17664.591,E2 -17664.591} C_VEL
LIN {X 0,Y 270.263,Z 289.444,A -85,B 0,C 180,E1 -17667.911,E2 -17667.911} C_VEL
LIN {X 0,Y 270.176,Z 289.455,A -85,B 0,C 180,E1 -17671.35,E2 -17671.35} C_VEL
LIN {X 0,Y 270.194,Z 289.455,A -85,B 0,C 180,E1 -17674.908,E2 -17674.908} C_VEL
LIN {X 0,Y 270.191,Z 289.455,A -85,B 0,C 180,E1 -17678.713,E2 -17678.713} C_VEL
LIN {X 0,Y 270.166,Z 289.455,A -85,B 0,C 180,E1 -17683.253,E2 -17683.253} C_VEL
LIN {X 0,Y 270.202,Z 289.502,A -85,B 0,C 180,E1 -17686.891,E2 -17686.891} C_VEL
LIN {X 0,Y 273.646,Z 303.561,A -85,B 0,C 180,E1 -17690.898,E2 -17690.898} C_VEL
LIN {X 0,Y 274.958,Z 308.875,A -85,B 0,C 180,E1 -17692.312,E2 -17692.312} C_VEL
LIN {X 0,Y 286.496,Z 340.082,A -85,B 0,C 180,E1 -17694.675,E2 -17694.675} C_VEL
LIN {X 0,Y 289.891,Z 368.142,A -85,B 0,C 180,E1 -17696.113,E2 -17696.113} C_VEL
LIN {X 0,Y 283.325,Z 476.442,A -85,B 0,C 180,E1 -17700.157,E2 -17700.157} C_VEL
LIN {X 0,Y 281.865,Z 493.013,A -85,B 0,C 180,E1 -17701.065,E2 -17701.065} C_VEL
LIN {X 0,Y 280.098,Z 508.987,A -85,B 0,C 180,E1 -17702.243,E2 -17702.243} C_VEL
LIN {X 0,Y 278.389,Z 523.199,A -85,B 0,C 180,E1 -17703.583,E2 -17703.583} C_VEL
LIN {X 0,Y 276.53,Z 537.188,A -85,B 0,C 180,E1 -17705.209,E2 -17705.209} C_VEL
LIN {X 0,Y 274.646,Z 550.555,A -85,B 0,C 180,E1 -17707.106,E2 -17707.106} C_VEL
LIN {X 0,Y 272.9,Z 563.122,A -85,B 0,C 180,E1 -17709.264,E2 -17709.264} C_VEL
LIN {X 0,Y 271.462,Z 574.014,A -85,B 0,C 180,E1 -17711.512,E2 -17711.512} C_VEL
LIN {X 0,Y 270.287,Z 583.956,A -85,B 0,C 180,E1 -17713.969,E2 -17713.969} C_VEL
LIN {X 0,Y 269.322,Z 593.41,A -85,B 0,C 180,E1 -17716.803,E2 -17716.803} C_VEL
LIN {X 0,Y 268.837,Z 600.579,A -85,B 0,C 180,E1 -17719.458,E2 -17719.458} C_VEL
LIN {X 0,Y 268.677,Z 605.589,A -85,B 0,C 180,E1 -17721.73,E2 -17721.73} C_VEL
LIN {X 0,Y 268.669,Z 609.695,A -85,B 0,C 180,E1 -17723.996,E2 -17723.996} C_VEL
LIN {X 0,Y 268.539,Z 613.729,A -85,B 0,C 180,E1 -17727.002,E2 -17727.002} C_VEL
LIN {X 0,Y 268.768,Z 615.223,A -85,B 0,C 180,E1 -17728.504,E2 -17728.504} C_VEL
LIN {X 0,Y 268.78,Z 616.33,A -85,B 0,C 180,E1 -17730.002,E2 -17730.002} C_VEL
LIN {X 0,Y 268.367,Z 617.493,A -85,B 0,C 180,E1 -17733.004,E2 -17733.004} C_VEL
LIN {X 0,Y 268.297,Z 617.394,A -85,B 0,C 180,E1 -17736.016,E2 -17736.016} C_VEL
LIN {X 0,Y 268.388,Z 616.061,A -85,B 0,C 180,E1 -17739.042,E2 -17739.042} C_VEL
LIN {X 0,Y 268.981,Z 613.52,A -85,B 0,C 180,E1 -17742.067,E2 -17742.067} C_VEL
LIN {X 0,Y 270.236,Z 609.75,A -85,B 0,C 180,E1 -17745.076,E2 -17745.076} C_VEL
LIN {X 0,Y 272.173,Z 604.764,A -85,B 0,C 180,E1 -17748.053,E2 -17748.053} C_VEL
LIN {X 0,Y 274.893,Z 598.488,A -85,B 0,C 180,E1 -17750.975,E2 -17750.975} C_VEL
LIN {X 0,Y 278.664,Z 589.816,A -85,B 0,C 180,E1 -17754.196,E2 -17754.196} C_VEL
LIN {X 0,Y 283.092,Z 580.457,A -85,B 0,C 180,E1 -17756.943,E2 -17756.943} C_VEL
LIN {X 0,Y 287.557,Z 570.874,A -85,B 0,C 180,E1 -17759.264,E2 -17759.264} C_VEL
LIN {X 0,Y 292.653,Z 559.805,A -85,B 0,C 180,E1 -17761.49,E2 -17761.49} C_VEL
LIN {X 0,Y 298.418,Z 546.915,A -85,B 0,C 180,E1 -17763.605,E2 -17763.605} C_VEL
LIN {X 0,Y 303.914,Z 534.099,A -85,B 0,C 180,E1 -17765.32,E2 -17765.32} C_VEL
LIN {X 0,Y 310.518,Z 517.779,A -85,B 0,C 180,E1 -17767.059,E2 -17767.059} C_VEL
LIN {X 0,Y 316.062,Z 502.793,A -85,B 0,C 180,E1 -17768.306,E2 -17768.306} C_VEL
LIN {X 0,Y 321.653,Z 485.644,A -85,B 0,C 180,E1 -17769.422,E2 -17769.422} C_VEL
LIN {X 0,Y 326.867,Z 466.63,A -85,B 0,C 180,E1 -17770.372,E2 -17770.372} C_VEL
LIN {X 0,Y 344.799,Z 387.488,A -85,B 0,C 180,E1 -17773.51,E2 -17773.51} C_VEL
LIN {X 0,Y 344.822,Z 385.797,A -85,B 0,C 180,E1 -17774.25,E2 -17774.25} C_VEL
LIN {X 0,Y 345.052,Z 383.691,A -85,B 0,C 180,E1 -17775.604,E2 -17775.604} C_VEL
LIN {X 0,Y 345.461,Z 383.717,A -85,B 0,C 180,E1 -17777.301,E2 -17777.301} C_VEL
LIN {X 0,Y 328.422,Z 457.106,A -85,B 0,C 180,E1 -17780.259,E2 -17780.259} C_VEL
LIN {X 0,Y 324.501,Z 472.064,A -85,B 0,C 180,E1 -17781.091,E2 -17781.091} C_VEL
LIN {X 0,Y 319.77,Z 487.415,A -85,B 0,C 180,E1 -17782.218,E2 -17782.218} C_VEL
LIN {X 0,Y 314.459,Z 502.407,A -85,B 0,C 180,E1 -17783.602,E2 -17783.602} C_VEL
LIN {X 0,Y 309.12,Z 516.129,A -85,B 0,C 180,E1 -17785.201,E2 -17785.201} C_VEL
LIN {X 0,Y 304.138,Z 527.732,A -85,B 0,C 180,E1 -17786.832,E2 -17786.832} C_VEL
LIN {X 0,Y 298.761,Z 539.425,A -85,B 0,C 180,E1 -17788.833,E2 -17788.833} C_VEL
LIN {X 0,Y 293.518,Z 549.935,A -85,B 0,C 180,E1 -17790.995,E2 -17790.995} C_VEL
LIN {X 0,Y 288.87,Z 558.817,A -85,B 0,C 180,E1 -17793.25,E2 -17793.25} C_VEL
LIN {X 0,Y 284.295,Z 567.31,A -85,B 0,C 180,E1 -17795.926,E2 -17795.926} C_VEL
LIN {X 0,Y 280.231,Z 574.329,A -85,B 0,C 180,E1 -17798.675,E2 -17798.675} C_VEL
LIN {X 0,Y 276.743,Z 579.956,A -85,B 0,C 180,E1 -17801.491,E2 -17801.491} C_VEL
LIN {X 0,Y 274.735,Z 583.287,A -85,B 0,C 180,E1 -17803.656,E2 -17803.656} C_VEL
LIN {X 0,Y 273.426,Z 585.157,A -85,B 0,C 180,E1 -17805.105,E2 -17805.105} C_VEL
LIN {X 0,Y 271.701,Z 587.901,A -85,B 0,C 180,E1 -17808.056,E2 -17808.056} C_VEL
LIN {X 0,Y 270.17,Z 589.5,A -85,B 0,C 180,E1 -17811.019,E2 -17811.019} C_VEL
LIN {X 0,Y 269.199,Z 589.925,A -85,B 0,C 180,E1 -17814.005,E2 -17814.005} C_VEL
LIN {X 0,Y 268.75,Z 589.161,A -85,B 0,C 180,E1 -17817.001,E2 -17817.001} C_VEL
LIN {X 0,Y 268.423,Z 587.2,A -85,B 0,C 180,E1 -17819.999,E2 -17819.999} C_VEL
LIN {X 0,Y 268.481,Z 583.977,A -85,B 0,C 180,E1 -17823,E2 -17823} C_VEL
LIN {X 0,Y 268.583,Z 579.248,A -85,B 0,C 180,E1 -17826.083,E2 -17826.083} C_VEL
LIN {X 0,Y 268.981,Z 573.317,A -85,B 0,C 180,E1 -17829.018,E2 -17829.018} C_VEL
LIN {X 0,Y 269.486,Z 566.657,A -85,B 0,C 180,E1 -17831.659,E2 -17831.659} C_VEL
LIN {X 0,Y 270.521,Z 558.573,A -85,B 0,C 180,E1 -17834.287,E2 -17834.287} C_VEL
LIN {X 0,Y 271.638,Z 548.967,A -85,B 0,C 180,E1 -17836.881,E2 -17836.881} C_VEL
LIN {X 0,Y 272.985,Z 538.85,A -85,B 0,C 180,E1 -17839.161,E2 -17839.161} C_VEL
LIN {X 0,Y 274.632,Z 527.103,A -85,B 0,C 180,E1 -17841.386,E2 -17841.386} C_VEL
LIN {X 0,Y 276.277,Z 514.046,A -85,B 0,C 180,E1 -17843.448,E2 -17843.448} C_VEL
LIN {X 0,Y 278.164,Z 500.31,A -85,B 0,C 180,E1 -17845.235,E2 -17845.235} C_VEL
LIN {X 0,Y 279.721,Z 486.878,A -85,B 0,C 180,E1 -17846.685,E2 -17846.685} C_VEL
LIN {X 0,Y 281.339,Z 471.389,A -85,B 0,C 180,E1 -17848.029,E2 -17848.029} C_VEL
LIN {X 0,Y 282.704,Z 454.712,A -85,B 0,C 180,E1 -17849.149,E2 -17849.149} C_VEL
LIN {X 0,Y 283.813,Z 438.438,A -85,B 0,C 180,E1 -17849.935,E2 -17849.935} C_VEL
LIN {X 0,Y 290.007,Z 335.37,A -85,B 0,C 180,E1 -17853.72,E2 -17853.72} C_VEL
LIN {X 0,Y 275.52,Z 301.982,A -85,B 0,C 180,E1 -17856.378,E2 -17856.378} C_VEL
LIN {X 0,Y 270.38,Z 290.203,A -85,B 0,C 180,E1 -17857.389,E2 -17857.389} C_VEL
LIN {X 0,Y 270.228,Z 289.451,A -85,B 0,C 180,E1 -17857.459,E2 -17857.459} C_VEL
LIN {X 0,Y 270.169,Z 289.456,A -85,B 0,C 180,E1 -17861.026,E2 -17861.026} C_VEL
LIN {X 0,Y 270.153,Z 289.459,A -85,B 0,C 180,E1 -17865.378,E2 -17865.378} C_VEL
LIN {X 0,Y 270.174,Z 289.456,A -85,B 0,C 180,E1 -17869.432,E2 -17869.432} C_VEL
LIN {X 0,Y 270.226,Z 289.451,A -85,B 0,C 180,E1 -17873.728,E2 -17873.728} C_VEL
LIN {X 0,Y 270.199,Z 289.451,A -85,B 0,C 180,E1 -17876.89,E2 -17876.89} C_VEL
LIN {X 0,Y 270.181,Z 289.453,A -85,B 0,C 180,E1 -17880.379,E2 -17880.379} C_VEL
LIN {X 0,Y 270.2,Z 289.454,A -85,B 0,C 180,E1 -17883.755,E2 -17883.755} C_VEL
LIN {X 0,Y 270.197,Z 289.451,A -85,B 0,C 180,E1 -17887.034,E2 -17887.034} C_VEL
LIN {X 0,Y 270.247,Z 289.446,A -85,B 0,C 180,E1 -17890.238,E2 -17890.238} C_VEL
LIN {X 0,Y 270.363,Z 289.432,A -85,B 0,C 180,E1 -17894.931,E2 -17894.931} C_VEL
LIN {X 0,Y 270.436,Z 289.425,A -85,B 0,C 180,E1 -17899.517,E2 -17899.517} C_VEL
LIN {X 0,Y 270.605,Z 289.4,A -85,B 0,C 180,E1 -17902.537,E2 -17902.537} C_VEL
LIN {X 0,Y 270.779,Z 289.378,A -85,B 0,C 180,E1 -17908.511,E2 -17908.511} C_VEL
LIN {X 0,Y 270.779,Z 289.381,A -85,B 0,C 180,E1 -17911.485,E2 -17911.485} C_VEL
LIN {X 0,Y 270.602,Z 289.405,A -85,B 0,C 180,E1 -17917.459,E2 -17917.459} C_VEL
LIN {X 0,Y 270.433,Z 289.42,A -85,B 0,C 180,E1 -17920.479,E2 -17920.479} C_VEL
LIN {X 0,Y 270.393,Z 289.428,A -85,B 0,C 180,E1 -17925.063,E2 -17925.063} C_VEL
LIN {X 0,Y 270.291,Z 289.441,A -85,B 0,C 180,E1 -17929.754,E2 -17929.754} C_VEL
LIN {X 0,Y 270.263,Z 289.442,A -85,B 0,C 180,E1 -17934.584,E2 -17934.584} C_VEL
LIN {X 0,Y 270.258,Z 289.443,A -85,B 0,C 180,E1 -17937.907,E2 -17937.907} C_VEL
LIN {X 0,Y 270.172,Z 289.458,A -85,B 0,C 180,E1 -17941.347,E2 -17941.347} C_VEL
LIN {X 0,Y 270.202,Z 289.45,A -85,B 0,C 180,E1 -17944.903,E2 -17944.903} C_VEL
LIN {X 0,Y 270.185,Z 289.453,A -85,B 0,C 180,E1 -17948.709,E2 -17948.709} C_VEL
LIN {X 0,Y 270.158,Z 289.459,A -85,B 0,C 180,E1 -17953.25,E2 -17953.25} C_VEL
LIN {X 0,Y 270.161,Z 289.458,A -85,B 0,C 180,E1 -17957.442,E2 -17957.442} C_VEL
LIN {X 0,Y 270.194,Z 289.453,A -85,B 0,C 180,E1 -17961.374,E2 -17961.374} C_VEL
LIN {X 0,Y 270.188,Z 289.455,A -85,B 0,C 180,E1 -17965.094,E2 -17965.094} C_VEL
LIN {X 0,Y 270.187,Z 289.456,A -85,B 0,C 180,E1 -17969.131,E2 -17969.131} C_VEL
LIN {X 0,Y 270.252,Z 289.443,A -85,B 0,C 180,E1 -17972.145,E2 -17972.145} C_VEL
LIN {X 0,Y 270.225,Z 289.449,A -85,B 0,C 180,E1 -17975.538,E2 -17975.538} C_VEL
LIN {X 0,Y 270.287,Z 289.438,A -85,B 0,C 180,E1 -17980.245,E2 -17980.245} C_VEL
LIN {X 0,Y 270.39,Z 289.43,A -85,B 0,C 180,E1 -17984.936,E2 -17984.936} C_VEL
LIN {X 0,Y 270.429,Z 289.423,A -85,B 0,C 180,E1 -17989.52,E2 -17989.52} C_VEL
LIN {X 0,Y 270.595,Z 289.402,A -85,B 0,C 180,E1 -17992.54,E2 -17992.54} C_VEL
LIN {X 0,Y 270.775,Z 289.379,A -85,B 0,C 180,E1 -17998.514,E2 -17998.514} C_VEL
LIN {X 0,Y 270.776,Z 289.379,A -85,B 0,C 180,E1 -18001.488,E2 -18001.488} C_VEL
LIN {X 0,Y 270.599,Z 289.402,A -85,B 0,C 180,E1 -18007.463,E2 -18007.463} C_VEL
LIN {X 0,Y 270.566,Z 289.407,A -85,B 0,C 180,E1 -18009.168,E2 -18009.168} C_VEL
LIN {X 0,Y 269.896,Z 289.49,A -85,B 0,C 180,E1 -18010.408,E2 -18010.408} C_VEL
LIN {X 0,Y 266.978,Z 289.853,A -85,B 0,C 180,E1 -18012.425,E2 -18012.425} C_VEL
LIN {X 0,Y 264.49,Z 290.164,A -85,B 0,C 180,E1 -18014.066,E2 -18014.066} C_VEL
LIN {X 0,Y 263.422,Z 290.297,A -85,B 0,C 180,E1 -18015.34,E2 -18015.34} C_VEL
LIN {X 0,Y 263.335,Z 290.306,A -85,B 0,C 180,E1 -18015.772,E2 -18015.772} C_VEL
LIN {X 0,Y 263.253,Z 290.318,A -85,B 0,C 180,E1 -18020.309,E2 -18020.309} C_VEL
LIN {X 0,Y 263.183,Z 290.327,A -85,B 0,C 180,E1 -18025.295,E2 -18025.295} C_VEL
LIN {X 0,Y 263.171,Z 290.331,A -85,B 0,C 180,E1 -18028.732,E2 -18028.732} C_VEL
LIN {X 0,Y 263.125,Z 290.333,A -85,B 0,C 180,E1 -18032.29,E2 -18032.29} C_VEL
LIN {X 0,Y 263.174,Z 290.33,A -85,B 0,C 180,E1 -18036.765,E2 -18036.765} C_VEL
LIN {X 0,Y 263.119,Z 290.331,A -85,B 0,C 180,E1 -18041.596,E2 -18041.596} C_VEL
LIN {X 0,Y 263.128,Z 290.331,A -85,B 0,C 180,E1 -18046.021,E2 -18046.021} C_VEL
LIN {X 0,Y 263.165,Z 290.515,A -85,B 0,C 180,E1 -18046.419,E2 -18046.419} C_VEL
LIN {X 0,Y 266.58,Z 304.436,A -85,B 0,C 180,E1 -18050.494,E2 -18050.494} C_VEL
LIN {X 0,Y 267.601,Z 308.505,A -85,B 0,C 180,E1 -18051.599,E2 -18051.599} C_VEL
LIN {X 0,Y 279.916,Z 341.892,A -85,B 0,C 180,E1 -18054.209,E2 -18054.209} C_VEL
LIN {X 0,Y 283.248,Z 368.544,A -85,B 0,C 180,E1 -18055.621,E2 -18055.621} C_VEL
LIN {X 0,Y 276.47,Z 476.329,A -85,B 0,C 180,E1 -18059.786,E2 -18059.786} C_VEL
LIN {X 0,Y 275.044,Z 492.097,A -85,B 0,C 180,E1 -18060.673,E2 -18060.673} C_VEL
LIN {X 0,Y 273.215,Z 508.339,A -85,B 0,C 180,E1 -18061.9,E2 -18061.9} C_VEL
LIN {X 0,Y 271.269,Z 524.264,A -85,B 0,C 180,E1 -18063.457,E2 -18063.457} C_VEL
LIN {X 0,Y 269.377,Z 537.963,A -85,B 0,C 180,E1 -18065.124,E2 -18065.124} C_VEL
LIN {X 0,Y 267.39,Z 551.9,A -85,B 0,C 180,E1 -18067.192,E2 -18067.192} C_VEL
LIN {X 0,Y 265.613,Z 564.536,A -85,B 0,C 180,E1 -18069.479,E2 -18069.479} C_VEL
LIN {X 0,Y 264.18,Z 575.137,A -85,B 0,C 180,E1 -18071.787,E2 -18071.787} C_VEL
LIN {X 0,Y 263.03,Z 585.473,A -85,B 0,C 180,E1 -18074.505,E2 -18074.505} C_VEL
LIN {X 0,Y 262.165,Z 593.988,A -85,B 0,C 180,E1 -18077.225,E2 -18077.225} C_VEL
LIN {X 0,Y 261.739,Z 600.982,A -85,B 0,C 180,E1 -18079.951,E2 -18079.951} C_VEL
LIN {X 0,Y 261.634,Z 605.827,A -85,B 0,C 180,E1 -18082.284,E2 -18082.284} C_VEL
LIN {X 0,Y 261.614,Z 609.323,A -85,B 0,C 180,E1 -18084.308,E2 -18084.308} C_VEL
LIN {X 0,Y 261.499,Z 612.762,A -85,B 0,C 180,E1 -18086.921,E2 -18086.921} C_VEL
LIN {X 0,Y 261.712,Z 614.349,A -85,B 0,C 180,E1 -18088.463,E2 -18088.463} C_VEL
LIN {X 0,Y 261.728,Z 615.549,A -85,B 0,C 180,E1 -18090.002,E2 -18090.002} C_VEL
LIN {X 0,Y 261.294,Z 616.889,A -85,B 0,C 180,E1 -18093.086,E2 -18093.086} C_VEL
LIN {X 0,Y 261.216,Z 616.978,A -85,B 0,C 180,E1 -18096.18,E2 -18096.18} C_VEL
LIN {X 0,Y 261.314,Z 615.794,A -85,B 0,C 180,E1 -18099.288,E2 -18099.288} C_VEL
LIN {X 0,Y 261.995,Z 613.416,A -85,B 0,C 180,E1 -18102.394,E2 -18102.394} C_VEL
LIN {X 0,Y 263.344,Z 609.882,A -85,B 0,C 180,E1 -18105.48,E2 -18105.48} C_VEL
LIN {X 0,Y 265.425,Z 605.162,A -85,B 0,C 180,E1 -18108.528,E2 -18108.528} C_VEL
LIN {X 0,Y 268.299,Z 599.187,A -85,B 0,C 180,E1 -18111.516,E2 -18111.516} C_VEL
LIN {X 0,Y 272.272,Z 590.88,A -85,B 0,C 180,E1 -18114.802,E2 -18114.802} C_VEL
LIN {X 0,Y 277.556,Z 580.674,A -85,B 0,C 180,E1 -18117.935,E2 -18117.935} C_VEL
LIN {X 0,Y 282.322,Z 571.372,A -85,B 0,C 180,E1 -18120.273,E2 -18120.273} C_VEL
LIN {X 0,Y 287.717,Z 560.627,A -85,B 0,C 180,E1 -18122.508,E2 -18122.508} C_VEL
LIN {X 0,Y 293.8,Z 548.153,A -85,B 0,C 180,E1 -18124.621,E2 -18124.621} C_VEL
LIN {X 0,Y 300.056,Z 534.727,A -85,B 0,C 180,E1 -18126.467,E2 -18126.467} C_VEL
LIN {X 0,Y 306.972,Z 518.87,A -85,B 0,C 180,E1 -18128.183,E2 -18128.183} C_VEL
LIN {X 0,Y 312.746,Z 504.488,A -85,B 0,C 180,E1 -18129.409,E2 -18129.409} C_VEL
LIN {X 0,Y 318.896,Z 487.332,A -85,B 0,C 180,E1 -18130.554,E2 -18130.554} C_VEL
LIN {X 0,Y 324.634,Z 468.149,A -85,B 0,C 180,E1 -18131.531,E2 -18131.531} C_VEL
LIN {X 0,Y 342.945,Z 392.435,A -85,B 0,C 180,E1 -18134.516,E2 -18134.516} C_VEL
LIN {X 0,Y 343.248,Z 390.488,A -85,B 0,C 180,E1 -18135.778,E2 -18135.778} C_VEL
LIN {X 0,Y 343.335,Z 390.423,A -85,B 0,C 180,E1 -18136.365,E2 -18136.365} C_VEL
LIN {X 0,Y 326.595,Z 458.376,A -85,B 0,C 180,E1 -18139.081,E2 -18139.081} C_VEL
LIN {X 0,Y 322.192,Z 473.851,A -85,B 0,C 180,E1 -18139.947,E2 -18139.947} C_VEL
LIN {X 0,Y 317.214,Z 488.771,A -85,B 0,C 180,E1 -18141.048,E2 -18141.048} C_VEL
LIN {X 0,Y 311.41,Z 503.947,A -85,B 0,C 180,E1 -18142.457,E2 -18142.457} C_VEL
LIN {X 0,Y 305.774,Z 517.217,A -85,B 0,C 180,E1 -18144.017,E2 -18144.017} C_VEL
LIN {X 0,Y 300.026,Z 529.61,A -85,B 0,C 180,E1 -18145.792,E2 -18145.792} C_VEL
LIN {X 0,Y 294.089,Z 541.454,A -85,B 0,C 180,E1 -18147.877,E2 -18147.877} C_VEL
LIN {X 0,Y 288.54,Z 551.628,A -85,B 0,C 180,E1 -18150.044,E2 -18150.044} C_VEL
LIN {X 0,Y 282.955,Z 561.37,A -85,B 0,C 180,E1 -18152.644,E2 -18152.644} C_VEL
LIN {X 0,Y 278.136,Z 569.436,A -85,B 0,C 180,E1 -18155.359,E2 -18155.359} C_VEL
LIN {X 0,Y 273.844,Z 576.114,A -85,B 0,C 180,E1 -18158.152,E2 -18158.152} C_VEL
LIN {X 0,Y 270.194,Z 581.454,A -85,B 0,C 180,E1 -18161.025,E2 -18161.025} C_VEL
LIN {X 0,Y 268.038,Z 584.548,A -85,B 0,C 180,E1 -18163.235,E2 -18163.235} C_VEL
LIN {X 0,Y 265.679,Z 587.682,A -85,B 0,C 180,E1 -18166.226,E2 -18166.226} C_VEL
LIN {X 0,Y 263.972,Z 589.657,A -85,B 0,C 180,E1 -18169.258,E2 -18169.258} C_VEL
LIN {X 0,Y 262.605,Z 590.488,A -85,B 0,C 180,E1 -18172.309,E2 -18172.309} C_VEL
LIN {X 0,Y 261.868,Z 590.101,A -85,B 0,C 180,E1 -18175.381,E2 -18175.381} C_VEL
LIN {X 0,Y 261.473,Z 588.536,A -85,B 0,C 180,E1 -18178.459,E2 -18178.459} C_VEL
LIN {X 0,Y 261.335,Z 585.744,A -85,B 0,C 180,E1 -18181.54,E2 -18181.54} C_VEL
LIN {X 0,Y 261.397,Z 581.643,A -85,B 0,C 180,E1 -18184.625,E2 -18184.625} C_VEL
LIN {X 0,Y 261.696,Z 576.12,A -85,B 0,C 180,E1 -18187.716,E2 -18187.716} C_VEL
LIN {X 0,Y 262.206,Z 569,A -85,B 0,C 180,E1 -18190.813,E2 -18190.813} C_VEL
LIN {X 0,Y 263.1,Z 561.319,A -85,B 0,C 180,E1 -18193.516,E2 -18193.516} C_VEL
LIN {X 0,Y 264.129,Z 552.245,A -85,B 0,C 180,E1 -18196.16,E2 -18196.16} C_VEL
LIN {X 0,Y 265.417,Z 542.561,A -85,B 0,C 180,E1 -18198.525,E2 -18198.525} C_VEL
LIN {X 0,Y 267.112,Z 530.39,A -85,B 0,C 180,E1 -18201.006,E2 -18201.006} C_VEL
LIN {X 0,Y 268.821,Z 518.131,A -85,B 0,C 180,E1 -18203.087,E2 -18203.087} C_VEL
LIN {X 0,Y 270.6,Z 504.902,A -85,B 0,C 180,E1 -18204.962,E2 -18204.962} C_VEL
LIN {X 0,Y 272.392,Z 490.588,A -85,B 0,C 180,E1 -18206.633,E2 -18206.633} C_VEL
LIN {X 0,Y 274.126,Z 474.909,A -85,B 0,C 180,E1 -18208.104,E2 -18208.104} C_VEL
LIN {X 0,Y 275.562,Z 458.657,A -85,B 0,C 180,E1 -18209.294,E2 -18209.294} C_VEL
LIN {X 0,Y 276.816,Z 441.96,A -85,B 0,C 180,E1 -18210.183,E2 -18210.183} C_VEL
LIN {X 0,Y 283.276,Z 337.084,A -85,B 0,C 180,E1 -18214.181,E2 -18214.181} C_VEL
LIN {X 0,Y 267.996,Z 301.884,A -85,B 0,C 180,E1 -18217.081,E2 -18217.081} C_VEL
LIN {X 0,Y 263.273,Z 290.91,A -85,B 0,C 180,E1 -18218.051,E2 -18218.051} C_VEL
LIN {X 0,Y 263.17,Z 290.331,A -85,B 0,C 180,E1 -18218.122,E2 -18218.122} C_VEL
LIN {X 0,Y 263.124,Z 290.337,A -85,B 0,C 180,E1 -18221.891,E2 -18221.891} C_VEL
LIN {X 0,Y 263.124,Z 290.335,A -85,B 0,C 180,E1 -18226.148,E2 -18226.148} C_VEL
LIN {X 0,Y 263.105,Z 290.335,A -85,B 0,C 180,E1 -18230.125,E2 -18230.125} C_VEL
LIN {X 0,Y 263.163,Z 290.329,A -85,B 0,C 180,E1 -18234.016,E2 -18234.016} C_VEL
LIN {X 0,Y 263.126,Z 290.336,A -85,B 0,C 180,E1 -18237.709,E2 -18237.709} C_VEL
LIN {X 0,Y 263.147,Z 290.333,A -85,B 0,C 180,E1 -18241.802,E2 -18241.802} C_VEL
LIN {X 0,Y 263.186,Z 290.325,A -85,B 0,C 180,E1 -18245.215,E2 -18245.215} C_VEL
LIN {X 0,Y 263.231,Z 290.324,A -85,B 0,C 180,E1 -18249.689,E2 -18249.689} C_VEL
LIN {X 0,Y 263.305,Z 290.311,A -85,B 0,C 180,E1 -18254.517,E2 -18254.517} C_VEL
LIN {X 0,Y 263.368,Z 290.304,A -85,B 0,C 180,E1 -18259.232,E2 -18259.232} C_VEL
LIN {X 0,Y 263.566,Z 290.277,A -85,B 0,C 180,E1 -18262.336,E2 -18262.336} C_VEL
LIN {X 0,Y 263.744,Z 290.255,A -85,B 0,C 180,E1 -18268.471,E2 -18268.471} C_VEL
LIN {X 0,Y 263.744,Z 290.257,A -85,B 0,C 180,E1 -18271.525,E2 -18271.525} C_VEL
LIN {X 0,Y 263.564,Z 290.28,A -85,B 0,C 180,E1 -18277.66,E2 -18277.66} C_VEL
LIN {X 0,Y 263.365,Z 290.3,A -85,B 0,C 180,E1 -18280.764,E2 -18280.764} C_VEL
LIN {X 0,Y 263.341,Z 290.309,A -85,B 0,C 180,E1 -18285.476,E2 -18285.476} C_VEL
LIN {X 0,Y 263.253,Z 290.315,A -85,B 0,C 180,E1 -18290.305,E2 -18290.305} C_VEL
LIN {X 0,Y 263.196,Z 290.326,A -85,B 0,C 180,E1 -18295.29,E2 -18295.29} C_VEL
LIN {X 0,Y 263.154,Z 290.328,A -85,B 0,C 180,E1 -18298.73,E2 -18298.73} C_VEL
LIN {X 0,Y 263.121,Z 290.332,A -85,B 0,C 180,E1 -18302.287,E2 -18302.287} C_VEL
LIN {X 0,Y 263.174,Z 290.325,A -85,B 0,C 180,E1 -18305.977,E2 -18305.977} C_VEL
LIN {X 0,Y 263.093,Z 290.336,A -85,B 0,C 180,E1 -18309.872,E2 -18309.872} C_VEL
LIN {X 0,Y 263.115,Z 290.331,A -85,B 0,C 180,E1 -18313.982,E2 -18313.982} C_VEL
LIN {X 0,Y 263.112,Z 290.333,A -85,B 0,C 180,E1 -18318.406,E2 -18318.406} C_VEL
LIN {X 0,Y 263.169,Z 290.329,A -85,B 0,C 180,E1 -18323.236,E2 -18323.236} C_VEL
LIN {X 0,Y 263.119,Z 290.333,A -85,B 0,C 180,E1 -18327.712,E2 -18327.712} C_VEL
LIN {X 0,Y 263.188,Z 290.323,A -85,B 0,C 180,E1 -18331.783,E2 -18331.783} C_VEL
LIN {X 0,Y 263.188,Z 290.328,A -85,B 0,C 180,E1 -18335.212,E2 -18335.212} C_VEL
LIN {X 0,Y 263.249,Z 290.316,A -85,B 0,C 180,E1 -18339.694,E2 -18339.694} C_VEL
LIN {X 0,Y 263.338,Z 290.306,A -85,B 0,C 180,E1 -18344.523,E2 -18344.523} C_VEL
LIN {X 0,Y 263.361,Z 290.305,A -85,B 0,C 180,E1 -18349.235,E2 -18349.235} C_VEL
LIN {X 0,Y 263.557,Z 290.278,A -85,B 0,C 180,E1 -18352.339,E2 -18352.339} C_VEL
LIN {X 0,Y 263.739,Z 290.256,A -85,B 0,C 180,E1 -18358.474,E2 -18358.474} C_VEL
LIN {X 0,Y 263.74,Z 290.256,A -85,B 0,C 180,E1 -18361.528,E2 -18361.528} C_VEL
LIN {X 0,Y 263.561,Z 290.278,A -85,B 0,C 180,E1 -18367.663,E2 -18367.663} C_VEL
LIN {X 0,Y 263.364,Z 290.305,A -85,B 0,C 180,E1 -18370.767,E2 -18370.767} C_VEL
LIN {X 0,Y 263.335,Z 290.306,A -85,B 0,C 180,E1 -18375.772,E2 -18375.772} C_VEL
LIN {X 0,Y 262.644,Z 290.396,A -85,B 0,C 180,E1 -18377.047,E2 -18377.047} C_VEL
LIN {X 0,Y 259.703,Z 290.762,A -85,B 0,C 180,E1 -18379.122,E2 -18379.122} C_VEL
LIN {X 0,Y 257.213,Z 291.074,A -85,B 0,C 180,E1 -18380.81,E2 -18380.81} C_VEL
LIN {X 0,Y 256.154,Z 291.202,A -85,B 0,C 180,E1 -18382.122,E2 -18382.122} C_VEL
LIN {X 0,Y 256.074,Z 291.214,A -85,B 0,C 180,E1 -18382.566,E2 -18382.566} C_VEL
LIN {X 0,Y 256.121,Z 291.206,A -85,B 0,C 180,E1 -18386.044,E2 -18386.044} C_VEL
LIN {X 0,Y 256.106,Z 291.207,A -85,B 0,C 180,E1 -18389.602,E2 -18389.602} C_VEL
LIN {X 0,Y 256.06,Z 291.213,A -85,B 0,C 180,E1 -18393.295,E2 -18393.295} C_VEL
LIN {X 0,Y 256.107,Z 291.207,A -85,B 0,C 180,E1 -18397.273,E2 -18397.273} C_VEL
LIN {X 0,Y 256.049,Z 291.213,A -85,B 0,C 180,E1 -18401.206,E2 -18401.206} C_VEL
LIN {X 0,Y 256.061,Z 291.212,A -85,B 0,C 180,E1 -18405.531,E2 -18405.531} C_VEL
LIN {X 0,Y 256.114,Z 291.452,A -85,B 0,C 180,E1 -18405.92,E2 -18405.92} C_VEL
LIN {X 0,Y 259.423,Z 304.798,A -85,B 0,C 180,E1 -18409.937,E2 -18409.937} C_VEL
LIN {X 0,Y 260.238,Z 308.166,A -85,B 0,C 180,E1 -18410.859,E2 -18410.859} C_VEL
LIN {X 0,Y 272.843,Z 342.309,A -85,B 0,C 180,E1 -18413.626,E2 -18413.626} C_VEL
LIN {X 0,Y 273.807,Z 346.036,A -85,B 0,C 180,E1 -18413.876,E2 -18413.876} C_VEL
LIN {X 0,Y 276.549,Z 369.688,A -85,B 0,C 180,E1 -18415.151,E2 -18415.151} C_VEL
LIN {X 0,Y 269.611,Z 476.112,A -85,B 0,C 180,E1 -18419.408,E2 -18419.408} C_VEL
LIN {X 0,Y 268.117,Z 492.248,A -85,B 0,C 180,E1 -18420.349,E2 -18420.349} C_VEL
LIN {X 0,Y 266.362,Z 507.584,A -85,B 0,C 180,E1 -18421.54,E2 -18421.54} C_VEL
LIN {X 0,Y 264.367,Z 523.513,A -85,B 0,C 180,E1 -18423.135,E2 -18423.135} C_VEL
LIN {X 0,Y 262.423,Z 537.226,A -85,B 0,C 180,E1 -18424.842,E2 -18424.842} C_VEL
LIN {X 0,Y 260.564,Z 550.118,A -85,B 0,C 180,E1 -18426.79,E2 -18426.79} C_VEL
LIN {X 0,Y 258.732,Z 562.883,A -85,B 0,C 180,E1 -18429.116,E2 -18429.116} C_VEL
LIN {X 0,Y 257.148,Z 574.514,A -85,B 0,C 180,E1 -18431.684,E2 -18431.684} C_VEL
LIN {X 0,Y 255.955,Z 584.887,A -85,B 0,C 180,E1 -18434.474,E2 -18434.474} C_VEL
LIN {X 0,Y 255.09,Z 593.416,A -85,B 0,C 180,E1 -18437.269,E2 -18437.269} C_VEL
LIN {X 0,Y 254.733,Z 599.486,A -85,B 0,C 180,E1 -18439.671,E2 -18439.671} C_VEL
LIN {X 0,Y 254.594,Z 606.011,A -85,B 0,C 180,E1 -18442.867,E2 -18442.867} C_VEL
LIN {X 0,Y 254.497,Z 609.755,A -85,B 0,C 180,E1 -18445.25,E2 -18445.25} C_VEL
LIN {X 0,Y 254.658,Z 613.454,A -85,B 0,C 180,E1 -18448.421,E2 -18448.421} C_VEL
LIN {X 0,Y 254.677,Z 614.752,A -85,B 0,C 180,E1 -18450.002,E2 -18450.002} C_VEL
LIN {X 0,Y 254.224,Z 616.272,A -85,B 0,C 180,E1 -18453.172,E2 -18453.172} C_VEL
LIN {X 0,Y 254.137,Z 616.49,A -85,B 0,C 180,E1 -18456.353,E2 -18456.353} C_VEL
LIN {X 0,Y 254.256,Z 615.484,A -85,B 0,C 180,E1 -18459.549,E2 -18459.549} C_VEL
LIN {X 0,Y 255.021,Z 613.331,A -85,B 0,C 180,E1 -18462.739,E2 -18462.739} C_VEL
LIN {X 0,Y 256.473,Z 610.046,A -85,B 0,C 180,E1 -18465.906,E2 -18465.906} C_VEL
LIN {X 0,Y 258.685,Z 605.547,A -85,B 0,C 180,E1 -18469.029,E2 -18469.029} C_VEL
LIN {X 0,Y 261.7,Z 599.83,A -85,B 0,C 180,E1 -18472.086,E2 -18472.086} C_VEL
LIN {X 0,Y 265.363,Z 592.884,A -85,B 0,C 180,E1 -18475.074,E2 -18475.074} C_VEL
LIN {X 0,Y 270.811,Z 583.38,A -85,B 0,C 180,E1 -18478.271,E2 -18478.271} C_VEL
LIN {X 0,Y 275.683,Z 574.679,A -85,B 0,C 180,E1 -18480.657,E2 -18480.657} C_VEL
LIN {X 0,Y 281.196,Z 564.694,A -85,B 0,C 180,E1 -18482.931,E2 -18482.931} C_VEL
LIN {X 0,Y 287.411,Z 553.146,A -85,B 0,C 180,E1 -18485.076,E2 -18485.076} C_VEL
LIN {X 0,Y 293.774,Z 540.844,A -85,B 0,C 180,E1 -18486.948,E2 -18486.948} C_VEL
LIN {X 0,Y 300.766,Z 526.484,A -85,B 0,C 180,E1 -18488.689,E2 -18488.689} C_VEL
LIN {X 0,Y 307.747,Z 510.95,A -85,B 0,C 180,E1 -18490.178,E2 -18490.178} C_VEL
LIN {X 0,Y 314.722,Z 493.769,A -85,B 0,C 180,E1 -18491.42,E2 -18491.42} C_VEL
LIN {X 0,Y 320.673,Z 476.629,A -85,B 0,C 180,E1 -18492.373,E2 -18492.373} C_VEL
LIN {X 0,Y 325.202,Z 461.093,A -85,B 0,C 180,E1 -18493.063,E2 -18493.063} C_VEL
LIN {X 0,Y 340.826,Z 399.563,A -85,B 0,C 180,E1 -18495.461,E2 -18495.461} C_VEL
LIN {X 0,Y 340.868,Z 399.404,A -85,B 0,C 180,E1 -18495.491,E2 -18495.491} C_VEL
LIN {X 0,Y 325.489,Z 458.606,A -85,B 0,C 180,E1 -18497.826,E2 -18497.826} C_VEL
LIN {X 0,Y 321.338,Z 472.511,A -85,B 0,C 180,E1 -18498.577,E2 -18498.577} C_VEL
LIN {X 0,Y 316.046,Z 487.64,A -85,B 0,C 180,E1 -18499.634,E2 -18499.634} C_VEL
LIN {X 0,Y 309.872,Z 502.823,A -85,B 0,C 180,E1 -18500.995,E2 -18500.995} C_VEL
LIN {X 0,Y 304.239,Z 515.293,A -85,B 0,C 180,E1 -18502.4,E2 -18502.4} C_VEL
LIN {X 0,Y 297.666,Z 528.585,A -85,B 0,C 180,E1 -18504.242,E2 -18504.242} C_VEL
LIN {X 0,Y 291.237,Z 540.513,A -85,B 0,C 180,E1 -18506.287,E2 -18506.287} C_VEL
LIN {X 0,Y 284.489,Z 552.126,A -85,B 0,C 180,E1 -18508.748,E2 -18508.748} C_VEL
LIN {X 0,Y 278.44,Z 561.803,A -85,B 0,C 180,E1 -18511.342,E2 -18511.342} C_VEL
LIN {X 0,Y 273.198,Z 569.831,A -85,B 0,C 180,E1 -18514.066,E2 -18514.066} C_VEL
LIN {X 0,Y 268.602,Z 576.455,A -85,B 0,C 180,E1 -18516.89,E2 -18516.89} C_VEL
LIN {X 0,Y 264.496,Z 581.824,A -85,B 0,C 180,E1 -18519.791,E2 -18519.791} C_VEL
LIN {X 0,Y 261.356,Z 585.848,A -85,B 0,C 180,E1 -18522.794,E2 -18522.794} C_VEL
LIN {X 0,Y 258.838,Z 588.707,A -85,B 0,C 180,E1 -18525.854,E2 -18525.854} C_VEL
LIN {X 0,Y 257.032,Z 590.426,A -85,B 0,C 180,E1 -18528.964,E2 -18528.964} C_VEL
LIN {X 0,Y 255.579,Z 591.042,A -85,B 0,C 180,E1 -18532.096,E2 -18532.096} C_VEL
LIN {X 0,Y 254.816,Z 590.487,A -85,B 0,C 180,E1 -18535.253,E2 -18535.253} C_VEL
LIN {X 0,Y 254.394,Z 588.721,A -85,B 0,C 180,E1 -18538.416,E2 -18538.416} C_VEL
LIN {X 0,Y 254.258,Z 585.717,A -85,B 0,C 180,E1 -18541.583,E2 -18541.583} C_VEL
LIN {X 0,Y 254.304,Z 581.403,A -85,B 0,C 180,E1 -18544.754,E2 -18544.754} C_VEL
LIN {X 0,Y 254.628,Z 575.644,A -85,B 0,C 180,E1 -18547.931,E2 -18547.931} C_VEL
LIN {X 0,Y 255.174,Z 568.293,A -85,B 0,C 180,E1 -18551.115,E2 -18551.115} C_VEL
LIN {X 0,Y 256.143,Z 560.353,A -85,B 0,C 180,E1 -18553.89,E2 -18553.89} C_VEL
LIN {X 0,Y 257.169,Z 551.363,A -85,B 0,C 180,E1 -18556.506,E2 -18556.506} C_VEL
LIN {X 0,Y 258.576,Z 540.998,A -85,B 0,C 180,E1 -18559.034,E2 -18559.034} C_VEL
LIN {X 0,Y 260.226,Z 529.506,A -85,B 0,C 180,E1 -18561.381,E2 -18561.381} C_VEL
LIN {X 0,Y 261.967,Z 517.008,A -85,B 0,C 180,E1 -18563.518,E2 -18563.518} C_VEL
LIN {X 0,Y 263.818,Z 503.488,A -85,B 0,C 180,E1 -18565.438,E2 -18565.438} C_VEL
LIN {X 0,Y 265.669,Z 488.82,A -85,B 0,C 180,E1 -18567.149,E2 -18567.149} C_VEL
LIN {X 0,Y 267.397,Z 473.777,A -85,B 0,C 180,E1 -18568.555,E2 -18568.555} C_VEL
LIN {X 0,Y 268.781,Z 457.701,A -85,B 0,C 180,E1 -18569.733,E2 -18569.733} C_VEL
LIN {X 0,Y 270.054,Z 440.967,A -85,B 0,C 180,E1 -18570.631,E2 -18570.631} C_VEL
LIN {X 0,Y 276.591,Z 338.862,A -85,B 0,C 180,E1 -18574.648,E2 -18574.648} C_VEL
LIN {X 0,Y 260.488,Z 301.618,A -85,B 0,C 180,E1 -18577.814,E2 -18577.814} C_VEL
LIN {X 0,Y 256.268,Z 291.978,A -85,B 0,C 180,E1 -18578.703,E2 -18578.703} C_VEL
LIN {X 0,Y 256.126,Z 291.207,A -85,B 0,C 180,E1 -18578.788,E2 -18578.788} C_VEL
LIN {X 0,Y 256.062,Z 291.215,A -85,B 0,C 180,E1 -18583.325,E2 -18583.325} C_VEL
LIN {X 0,Y 256.072,Z 291.214,A -85,B 0,C 180,E1 -18587.817,E2 -18587.817} C_VEL
LIN {X 0,Y 256.071,Z 291.21,A -85,B 0,C 180,E1 -18590.856,E2 -18590.856} C_VEL
LIN {X 0,Y 256.131,Z 291.204,A -85,B 0,C 180,E1 -18592.865,E2 -18592.865} C_VEL
LIN {X 0,Y 256.064,Z 291.212,A -85,B 0,C 180,E1 -18596.705,E2 -18596.705} C_VEL
LIN {X 0,Y 256.053,Z 291.213,A -85,B 0,C 180,E1 -18600.391,E2 -18600.391} C_VEL
LIN {X 0,Y 256.13,Z 291.203,A -85,B 0,C 180,E1 -18604.886,E2 -18604.886} C_VEL
LIN {X 0,Y 256.143,Z 291.203,A -85,B 0,C 180,E1 -18609.101,E2 -18609.101} C_VEL
LIN {X 0,Y 256.226,Z 291.194,A -85,B 0,C 180,E1 -18614.078,E2 -18614.078} C_VEL
LIN {X 0,Y 256.284,Z 291.187,A -85,B 0,C 180,E1 -18617.325,E2 -18617.325} C_VEL
LIN {X 0,Y 256.475,Z 291.161,A -85,B 0,C 180,E1 -18620.558,E2 -18620.558} C_VEL
LIN {X 0,Y 256.48,Z 291.162,A -85,B 0,C 180,E1 -18623.705,E2 -18623.705} C_VEL
LIN {X 0,Y 256.707,Z 291.131,A -85,B 0,C 180,E1 -18628.429,E2 -18628.429} C_VEL
LIN {X 0,Y 256.706,Z 291.133,A -85,B 0,C 180,E1 -18631.567,E2 -18631.567} C_VEL
LIN {X 0,Y 256.531,Z 291.154,A -85,B 0,C 180,E1 -18637.871,E2 -18637.871} C_VEL
LIN {X 0,Y 256.301,Z 291.181,A -85,B 0,C 180,E1 -18641.064,E2 -18641.064} C_VEL
LIN {X 0,Y 256.29,Z 291.184,A -85,B 0,C 180,E1 -18645.913,E2 -18645.913} C_VEL
LIN {X 0,Y 256.157,Z 291.2,A -85,B 0,C 180,E1 -18650.893,E2 -18650.893} C_VEL
LIN {X 0,Y 256.177,Z 291.199,A -85,B 0,C 180,E1 -18655.137,E2 -18655.137} C_VEL
LIN {X 0,Y 256.092,Z 291.211,A -85,B 0,C 180,E1 -18659.6,E2 -18659.6} C_VEL
LIN {X 0,Y 256.073,Z 291.214,A -85,B 0,C 180,E1 -18663.289,E2 -18663.289} C_VEL
LIN {X 0,Y 256.115,Z 291.207,A -85,B 0,C 180,E1 -18667.273,E2 -18667.273} C_VEL
LIN {X 0,Y 256.06,Z 291.211,A -85,B 0,C 180,E1 -18672.181,E2 -18672.181} C_VEL
LIN {X 0,Y 256.052,Z 291.213,A -85,B 0,C 180,E1 -18676.673,E2 -18676.673} C_VEL
LIN {X 0,Y 256.058,Z 291.213,A -85,B 0,C 180,E1 -18680.858,E2 -18680.858} C_VEL
LIN {X 0,Y 256.117,Z 291.204,A -85,B 0,C 180,E1 -18682.867,E2 -18682.867} C_VEL
LIN {X 0,Y 256.054,Z 291.213,A -85,B 0,C 180,E1 -18686.707,E2 -18686.707} C_VEL
LIN {X 0,Y 256.101,Z 291.205,A -85,B 0,C 180,E1 -18690.4,E2 -18690.4} C_VEL
LIN {X 0,Y 256.158,Z 291.202,A -85,B 0,C 180,E1 -18694.87,E2 -18694.87} C_VEL
LIN {X 0,Y 256.149,Z 291.203,A -85,B 0,C 180,E1 -18699.105,E2 -18699.105} C_VEL
LIN {X 0,Y 256.287,Z 291.183,A -85,B 0,C 180,E1 -18704.086,E2 -18704.086} C_VEL
LIN {X 0,Y 256.297,Z 291.184,A -85,B 0,C 180,E1 -18708.935,E2 -18708.935} C_VEL
LIN {X 0,Y 256.525,Z 291.154,A -85,B 0,C 180,E1 -18712.128,E2 -18712.128} C_VEL
LIN {X 0,Y 256.702,Z 291.132,A -85,B 0,C 180,E1 -18718.432,E2 -18718.432} C_VEL
LIN {X 0,Y 256.703,Z 291.132,A -85,B 0,C 180,E1 -18721.57,E2 -18721.57} C_VEL
LIN {X 0,Y 256.529,Z 291.153,A -85,B 0,C 180,E1 -18727.874,E2 -18727.874} C_VEL
LIN {X 0,Y 256.299,Z 291.186,A -85,B 0,C 180,E1 -18731.068,E2 -18731.068} C_VEL
LIN {X 0,Y 256.29,Z 291.184,A -85,B 0,C 180,E1 -18735.917,E2 -18735.917} C_VEL
LIN {X 0,Y 256.153,Z 291.206,A -85,B 0,C 180,E1 -18740.897,E2 -18740.897} C_VEL
LIN {X 0,Y 256.074,Z 291.214,A -85,B 0,C 180,E1 -18742.566,E2 -18742.566} C_VEL
LIN {X 0,Y 255.428,Z 291.301,A -85,B 0,C 180,E1 -18743.879,E2 -18743.879} C_VEL
LIN {X 0,Y 252.609,Z 291.654,A -85,B 0,C 180,E1 -18746.021,E2 -18746.021} C_VEL
LIN {X 0,Y 250.193,Z 291.95,A -85,B 0,C 180,E1 -18747.763,E2 -18747.763} C_VEL
LIN {X 0,Y 249.138,Z 292.078,A -85,B 0,C 180,E1 -18749.114,E2 -18749.114} C_VEL
LIN {X 0,Y 249.043,Z 292.087,A -85,B 0,C 180,E1 -18749.572,E2 -18749.572} C_VEL
LIN {X 0,Y 249.023,Z 292.091,A -85,B 0,C 180,E1 -18752.428,E2 -18752.428} C_VEL
LIN {X 0,Y 249.04,Z 292.088,A -85,B 0,C 180,E1 -18756.345,E2 -18756.345} C_VEL
LIN {X 0,Y 249,Z 292.093,A -85,B 0,C 180,E1 -18760.48,E2 -18760.48} C_VEL
LIN {X 0,Y 249.004,Z 292.091,A -85,B 0,C 180,E1 -18764.88,E2 -18764.88} C_VEL
LIN {X 0,Y 249.024,Z 292.136,A -85,B 0,C 180,E1 -18765.33,E2 -18765.33} C_VEL
LIN {X 0,Y 252.28,Z 305.374,A -85,B 0,C 180,E1 -18769.43,E2 -18769.43} C_VEL
LIN {X 0,Y 252.821,Z 307.595,A -85,B 0,C 180,E1 -18770.087,E2 -18770.087} C_VEL
LIN {X 0,Y 266.03,Z 343.466,A -85,B 0,C 180,E1 -18773.083,E2 -18773.083} C_VEL
LIN {X 0,Y 267.315,Z 347.792,A -85,B 0,C 180,E1 -18773.397,E2 -18773.397} C_VEL
LIN {X 0,Y 269.896,Z 369.818,A -85,B 0,C 180,E1 -18774.63,E2 -18774.63} C_VEL
LIN {X 0,Y 262.838,Z 475.173,A -85,B 0,C 180,E1 -18778.99,E2 -18778.99} C_VEL
LIN {X 0,Y 261.289,Z 491.178,A -85,B 0,C 180,E1 -18779.939,E2 -18779.939} C_VEL
LIN {X 0,Y 259.526,Z 506.615,A -85,B 0,C 180,E1 -18781.163,E2 -18781.163} C_VEL
LIN {X 0,Y 257.484,Z 522.626,A -85,B 0,C 180,E1 -18782.797,E2 -18782.797} C_VEL
LIN {X 0,Y 255.499,Z 536.41,A -85,B 0,C 180,E1 -18784.548,E2 -18784.548} C_VEL
LIN {X 0,Y 253.621,Z 549.084,A -85,B 0,C 180,E1 -18786.504,E2 -18786.504} C_VEL
LIN {X 0,Y 251.826,Z 561.11,A -85,B 0,C 180,E1 -18788.73,E2 -18788.73} C_VEL
LIN {X 0,Y 250.341,Z 572.11,A -85,B 0,C 180,E1 -18791.167,E2 -18791.167} C_VEL
LIN {X 0,Y 249.196,Z 581.409,A -85,B 0,C 180,E1 -18793.621,E2 -18793.621} C_VEL
LIN {X 0,Y 248.231,Z 590.484,A -85,B 0,C 180,E1 -18796.495,E2 -18796.495} C_VEL
LIN {X 0,Y 247.714,Z 597.922,A -85,B 0,C 180,E1 -18799.375,E2 -18799.375} C_VEL
LIN {X 0,Y 247.548,Z 603.185,A -85,B 0,C 180,E1 -18801.842,E2 -18801.842} C_VEL
LIN {X 0,Y 247.538,Z 607.249,A -85,B 0,C 180,E1 -18804.202,E2 -18804.202} C_VEL
LIN {X 0,Y 247.423,Z 610.757,A -85,B 0,C 180,E1 -18806.746,E2 -18806.746} C_VEL
LIN {X 0,Y 247.606,Z 612.525,A -85,B 0,C 180,E1 -18808.376,E2 -18808.376} C_VEL
LIN {X 0,Y 247.626,Z 613.901,A -85,B 0,C 180,E1 -18810.002,E2 -18810.002} C_VEL
LIN {X 0,Y 247.407,Z 614.897,A -85,B 0,C 180,E1 -18811.63,E2 -18811.63} C_VEL
LIN {X 0,Y 247.107,Z 616.004,A -85,B 0,C 180,E1 -18815.467,E2 -18815.467} C_VEL
LIN {X 0,Y 247.055,Z 615.719,A -85,B 0,C 180,E1 -18818.179,E2 -18818.179} C_VEL
LIN {X 0,Y 247.499,Z 614.363,A -85,B 0,C 180,E1 -18821.467,E2 -18821.467} C_VEL
LIN {X 0,Y 248.716,Z 611.834,A -85,B 0,C 180,E1 -18824.735,E2 -18824.735} C_VEL
LIN {X 0,Y 250.666,Z 608.163,A -85,B 0,C 180,E1 -18827.966,E2 -18827.966} C_VEL
LIN {X 0,Y 253.461,Z 603.366,A -85,B 0,C 180,E1 -18831.131,E2 -18831.131} C_VEL
LIN {X 0,Y 257.037,Z 597.388,A -85,B 0,C 180,E1 -18834.215,E2 -18834.215} C_VEL
LIN {X 0,Y 260.153,Z 592.063,A -85,B 0,C 180,E1 -18836.473,E2 -18836.473} C_VEL
LIN {X 0,Y 266.121,Z 582.63,A -85,B 0,C 180,E1 -18839.683,E2 -18839.683} C_VEL
LIN {X 0,Y 272.182,Z 572.712,A -85,B 0,C 180,E1 -18842.399,E2 -18842.399} C_VEL
LIN {X 0,Y 279.147,Z 561.11,A -85,B 0,C 180,E1 -18844.946,E2 -18844.946} C_VEL
LIN {X 0,Y 286.961,Z 547.543,A -85,B 0,C 180,E1 -18847.314,E2 -18847.314} C_VEL
LIN {X 0,Y 294.59,Z 533.543,A -85,B 0,C 180,E1 -18849.215,E2 -18849.215} C_VEL
LIN {X 0,Y 301.656,Z 519.582,A -85,B 0,C 180,E1 -18850.721,E2 -18850.721} C_VEL
LIN {X 0,Y 307.98,Z 506.046,A -85,B 0,C 180,E1 -18851.874,E2 -18851.874} C_VEL
LIN {X 0,Y 314.629,Z 490.077,A -85,B 0,C 180,E1 -18852.946,E2 -18852.946} C_VEL
LIN {X 0,Y 321.191,Z 471.652,A -85,B 0,C 180,E1 -18853.898,E2 -18853.898} C_VEL
LIN {X 0,Y 326.715,Z 452.486,A -85,B 0,C 180,E1 -18854.681,E2 -18854.681} C_VEL
LIN {X 0,Y 331.919,Z 432.678,A -85,B 0,C 180,E1 -18855.443,E2 -18855.443} C_VEL
LIN {X 0,Y 331.969,Z 432.492,A -85,B 0,C 180,E1 -18855.509,E2 -18855.509} C_VEL
LIN {X 0,Y 324.036,Z 461.671,A -85,B 0,C 180,E1 -18856.692,E2 -18856.692} C_VEL
LIN {X 0,Y 318.93,Z 477.126,A -85,B 0,C 180,E1 -18857.556,E2 -18857.556} C_VEL
LIN {X 0,Y 313.406,Z 491.321,A -85,B 0,C 180,E1 -18858.583,E2 -18858.583} C_VEL
LIN {X 0,Y 306.411,Z 507.04,A -85,B 0,C 180,E1 -18860.041,E2 -18860.041} C_VEL
LIN {X 0,Y 299.86,Z 520.167,A -85,B 0,C 180,E1 -18861.603,E2 -18861.603} C_VEL
LIN {X 0,Y 292.669,Z 533.246,A -85,B 0,C 180,E1 -18863.534,E2 -18863.534} C_VEL
LIN {X 0,Y 286.037,Z 544.385,A -85,B 0,C 180,E1 -18865.589,E2 -18865.589} C_VEL
LIN {X 0,Y 278.93,Z 555.345,A -85,B 0,C 180,E1 -18868.053,E2 -18868.053} C_VEL
LIN {X 0,Y 272.661,Z 564.477,A -85,B 0,C 180,E1 -18870.676,E2 -18870.676} C_VEL
LIN {X 0,Y 267.165,Z 572.068,A -85,B 0,C 180,E1 -18873.435,E2 -18873.435} C_VEL
LIN {X 0,Y 262.322,Z 578.315,A -85,B 0,C 180,E1 -18876.304,E2 -18876.304} C_VEL
LIN {X 0,Y 258.001,Z 583.355,A -85,B 0,C 180,E1 -18879.259,E2 -18879.259} C_VEL
LIN {X 0,Y 254.695,Z 587.121,A -85,B 0,C 180,E1 -18882.329,E2 -18882.329} C_VEL
LIN {X 0,Y 252.014,Z 589.753,A -85,B 0,C 180,E1 -18885.463,E2 -18885.463} C_VEL
LIN {X 0,Y 250.11,Z 591.205,A -85,B 0,C 180,E1 -18888.655,E2 -18888.655} C_VEL
LIN {X 0,Y 248.573,Z 591.57,A -85,B 0,C 180,E1 -18891.872,E2 -18891.872} C_VEL
LIN {X 0,Y 247.744,Z 590.781,A -85,B 0,C 180,E1 -18895.117,E2 -18895.117} C_VEL
LIN {X 0,Y 247.317,Z 588.829,A -85,B 0,C 180,E1 -18898.37,E2 -18898.37} C_VEL
LIN {X 0,Y 247.182,Z 585.645,A -85,B 0,C 180,E1 -18901.628,E2 -18901.628} C_VEL
LIN {X 0,Y 247.205,Z 582.345,A -85,B 0,C 180,E1 -18904.074,E2 -18904.074} C_VEL
LIN {X 0,Y 247.464,Z 576.736,A -85,B 0,C 180,E1 -18907.341,E2 -18907.341} C_VEL
LIN {X 0,Y 247.898,Z 570.544,A -85,B 0,C 180,E1 -18910.205,E2 -18910.205} C_VEL
LIN {X 0,Y 248.656,Z 562.975,A -85,B 0,C 180,E1 -18913.067,E2 -18913.067} C_VEL
LIN {X 0,Y 249.633,Z 555.28,A -85,B 0,C 180,E1 -18915.512,E2 -18915.512} C_VEL
LIN {X 0,Y 251.016,Z 544.577,A -85,B 0,C 180,E1 -18918.358,E2 -18918.358} C_VEL
LIN {X 0,Y 252.558,Z 533.648,A -85,B 0,C 180,E1 -18920.779,E2 -18920.779} C_VEL
LIN {X 0,Y 254.307,Z 521.841,A -85,B 0,C 180,E1 -18922.975,E2 -18922.975} C_VEL
LIN {X 0,Y 256.273,Z 507.576,A -85,B 0,C 180,E1 -18925.175,E2 -18925.175} C_VEL
LIN {X 0,Y 258.095,Z 493.863,A -85,B 0,C 180,E1 -18926.916,E2 -18926.916} C_VEL
LIN {X 0,Y 259.871,Z 478.864,A -85,B 0,C 180,E1 -18928.465,E2 -18928.465} C_VEL
LIN {X 0,Y 261.434,Z 463.691,A -85,B 0,C 180,E1 -18929.711,E2 -18929.711} C_VEL
LIN {X 0,Y 262.749,Z 446.731,A -85,B 0,C 180,E1 -18930.768,E2 -18930.768} C_VEL
LIN {X 0,Y 265.423,Z 406.311,A -85,B 0,C 180,E1 -18932.479,E2 -18932.479} C_VEL
LIN {X 0,Y 269.908,Z 340.672,A -85,B 0,C 180,E1 -18935.128,E2 -18935.128} C_VEL
LIN {X 0,Y 253.836,Z 303.41,A -85,B 0,C 180,E1 -18938.379,E2 -18938.379} C_VEL
LIN {X 0,Y 249.209,Z 292.942,A -85,B 0,C 180,E1 -18939.383,E2 -18939.383} C_VEL
LIN {X 0,Y 249.044,Z 292.09,A -85,B 0,C 180,E1 -18939.501,E2 -18939.501} C_VEL
LIN {X 0,Y 249.009,Z 292.093,A -85,B 0,C 180,E1 -18942.79,E2 -18942.79} C_VEL
LIN {X 0,Y 249.016,Z 292.092,A -85,B 0,C 180,E1 -18947.36,E2 -18947.36} C_VEL
LIN {X 0,Y 249.044,Z 292.088,A -85,B 0,C 180,E1 -18952.198,E2 -18952.198} C_VEL
LIN {X 0,Y 249.042,Z 292.089,A -85,B 0,C 180,E1 -18955.637,E2 -18955.637} C_VEL
LIN {X 0,Y 249,Z 292.092,A -85,B 0,C 180,E1 -18959.464,E2 -18959.464} C_VEL
LIN {X 0,Y 249.033,Z 292.088,A -85,B 0,C 180,E1 -18963.155,E2 -18963.155} C_VEL
LIN {X 0,Y 249.051,Z 292.085,A -85,B 0,C 180,E1 -18966.728,E2 -18966.728} C_VEL
LIN {X 0,Y 249.074,Z 292.084,A -85,B 0,C 180,E1 -18970.206,E2 -18970.206} C_VEL
LIN {X 0,Y 249.172,Z 292.075,A -85,B 0,C 180,E1 -18973.615,E2 -18973.615} C_VEL
LIN {X 0,Y 249.246,Z 292.061,A -85,B 0,C 180,E1 -18978.614,E2 -18978.614} C_VEL
LIN {X 0,Y 249.476,Z 292.035,A -85,B 0,C 180,E1 -18981.901,E2 -18981.901} C_VEL
LIN {X 0,Y 249.427,Z 292.039,A -85,B 0,C 180,E1 -18986.767,E2 -18986.767} C_VEL
LIN {X 0,Y 249.721,Z 292.002,A -85,B 0,C 180,E1 -18989.998,E2 -18989.998} C_VEL
LIN {X 0,Y 249.427,Z 292.039,A -85,B 0,C 180,E1 -18993.228,E2 -18993.228} C_VEL
LIN {X 0,Y 249.473,Z 292.032,A -85,B 0,C 180,E1 -18998.095,E2 -18998.095} C_VEL
LIN {X 0,Y 249.244,Z 292.062,A -85,B 0,C 180,E1 -19001.381,E2 -19001.381} C_VEL
LIN {X 0,Y 249.233,Z 292.062,A -85,B 0,C 180,E1 -19006.376,E2 -19006.376} C_VEL
LIN {X 0,Y 249.077,Z 292.085,A -85,B 0,C 180,E1 -19011.516,E2 -19011.516} C_VEL
LIN {X 0,Y 249.119,Z 292.078,A -85,B 0,C 180,E1 -19015.48,E2 -19015.48} C_VEL
LIN {X 0,Y 249.061,Z 292.084,A -85,B 0,C 180,E1 -19018.987,E2 -19018.987} C_VEL
LIN {X 0,Y 249.024,Z 292.088,A -85,B 0,C 180,E1 -19022.424,E2 -19022.424} C_VEL
LIN {X 0,Y 249.056,Z 292.082,A -85,B 0,C 180,E1 -19026.338,E2 -19026.338} C_VEL
LIN {X 0,Y 248.993,Z 292.092,A -85,B 0,C 180,E1 -19030.477,E2 -19030.477} C_VEL
LIN {X 0,Y 248.994,Z 292.091,A -85,B 0,C 180,E1 -19034.877,E2 -19034.877} C_VEL
LIN {X 0,Y 249.005,Z 292.094,A -85,B 0,C 180,E1 -19037.363,E2 -19037.363} C_VEL
LIN {X 0,Y 249.03,Z 292.085,A -85,B 0,C 180,E1 -19042.2,E2 -19042.2} C_VEL
LIN {X 0,Y 249.03,Z 292.089,A -85,B 0,C 180,E1 -19045.639,E2 -19045.639} C_VEL
LIN {X 0,Y 249.039,Z 292.087,A -85,B 0,C 180,E1 -19049.473,E2 -19049.473} C_VEL
LIN {X 0,Y 249.058,Z 292.087,A -85,B 0,C 180,E1 -19053.162,E2 -19053.162} C_VEL
LIN {X 0,Y 249.048,Z 292.086,A -85,B 0,C 180,E1 -19056.731,E2 -19056.731} C_VEL
LIN {X 0,Y 249.095,Z 292.078,A -85,B 0,C 180,E1 -19060.212,E2 -19060.212} C_VEL
LIN {X 0,Y 249.23,Z 292.064,A -85,B 0,C 180,E1 -19063.623,E2 -19063.623} C_VEL
LIN {X 0,Y 249.24,Z 292.06,A -85,B 0,C 180,E1 -19068.617,E2 -19068.617} C_VEL
LIN {X 0,Y 249.467,Z 292.033,A -85,B 0,C 180,E1 -19071.904,E2 -19071.904} C_VEL
LIN {X 0,Y 249.423,Z 292.041,A -85,B 0,C 180,E1 -19076.771,E2 -19076.771} C_VEL
LIN {X 0,Y 249.717,Z 292.002,A -85,B 0,C 180,E1 -19080.001,E2 -19080.001} C_VEL
LIN {X 0,Y 249.422,Z 292.041,A -85,B 0,C 180,E1 -19083.232,E2 -19083.232} C_VEL
